ABB RAPID module: ReplayTargets_v13.mod

MODULE ReplayTargets_v13
    ! Generated from tests_v13.csv and success_v13.csv.
    ! Target names include version and testId. B* variants include version, testId, and confId.

    ! Robtargets and jointtargets for replay
    CONST robtarget rA_v13_t1 := [[1867.5,0,1823],[2.18557E-8,0,-1,0],[0,0,0,0],[9E+09,9E+09,9E+09,9E+09,9E+09,9E+09]];
    CONST robtarget rB_v13_t1 := [[99.2091,-1417.11,3170.05],[0.75375,-0.215208,0.229423,-0.576985],[-2,-3,2,0],[9E+09,9E+09,9E+09,9E+09,9E+09,9E+09]];
    CONST robtarget rB_v13_t1_c2 := [[99.2091,-1417.11,3170.05],[0.75375,-0.215208,0.229423,-0.576985],[0,0,-4,0],[9E+09,9E+09,9E+09,9E+09,9E+09,9E+09]];
    CONST jointtarget jA_v13_t1 := [[0,-2.3802E-6,7.25062E-7,0,90,0],[9E+09,9E+09,9E+09,9E+09,9E+09,9E+09]];
    CONST jointtarget jB_v13_t1 := [[-90.0009,9.75799,-56.39,-225.001,57.1728,224.999],[9E+09,9E+09,9E+09,9E+09,9E+09,9E+09]];
    CONST jointtarget jBseed_v13_t1 := [[-90.0009,9.75799,-56.39,-225.001,57.1728,224.999],[9E+09,9E+09,9E+09,9E+09,9E+09,9E+09]];

    CONST robtarget rA_v13_t2 := [[99.2091,-1417.11,3170.05],[0.75375,-0.215208,0.229423,-0.576985],[-2,-3,2,0],[9E+09,9E+09,9E+09,9E+09,9E+09,9E+09]];
    CONST robtarget rB_v13_t2 := [[-1176.87,-1004.25,553.318],[0.0696016,-0.873055,0.122095,0.466929],[-2,3,1,0],[9E+09,9E+09,9E+09,9E+09,9E+09,9E+09]];
    CONST robtarget rB_v13_t2_c5 := [[-1176.87,-1004.25,553.318],[0.0696016,-0.873055,0.122095,0.466929],[0,0,0,0],[9E+09,9E+09,9E+09,9E+09,9E+09,9E+09]];
    CONST jointtarget jA_v13_t2 := [[-90.0009,9.75799,-56.39,-225.001,57.1728,224.999],[9E+09,9E+09,9E+09,9E+09,9E+09,9E+09]];
    CONST jointtarget jB_v13_t2 := [[-134.999,4.65286,49.6707,270.001,46.9753,135.001],[9E+09,9E+09,9E+09,9E+09,9E+09,9E+09]];
    CONST jointtarget jBseed_v13_t2 := [[-134.999,4.65285,49.6707,270.001,46.9753,135.001],[9E+09,9E+09,9E+09,9E+09,9E+09,9E+09]];

    CONST robtarget rA_v13_t3 := [[-1176.87,-1004.25,553.318],[0.0696016,-0.873055,0.122095,0.466929],[-2,3,1,0],[9E+09,9E+09,9E+09,9E+09,9E+09,9E+09]];
    CONST robtarget rB_v13_t3 := [[-0.00217641,-566.482,3480.85],[0.983173,-0.182676,1.08969E-6,-6.64925E-6],[-2,-3,-2,0],[9E+09,9E+09,9E+09,9E+09,9E+09,9E+09]];
    CONST robtarget rB_v13_t3_c8 := [[-0.00217641,-566.482,3480.85],[0.983173,-0.182676,1.08969E-6,-6.64925E-6],[0,0,4,0],[9E+09,9E+09,9E+09,9E+09,9E+09,9E+09]];
    CONST jointtarget jA_v13_t3 := [[-134.999,4.65286,49.6707,270.001,46.9753,135.001],[9E+09,9E+09,9E+09,9E+09,9E+09,9E+09]];
    CONST jointtarget jB_v13_t3 := [[-90.0003,1.44106,-73.8029,-180,38.6896,-90.0003],[9E+09,9E+09,9E+09,9E+09,9E+09,9E+09]];
    CONST jointtarget jBseed_v13_t3 := [[-90.0003,1.44108,-73.8029,-180,38.6895,-90.0003],[9E+09,9E+09,9E+09,9E+09,9E+09,9E+09]];

    CONST robtarget rA_v13_t4 := [[-0.00217641,-566.482,3480.85],[0.983173,-0.182676,1.08969E-6,-6.64925E-6],[-2,-3,-2,0],[9E+09,9E+09,9E+09,9E+09,9E+09,9E+09]];
    CONST robtarget rB_v13_t4 := [[1002.23,-1002.24,1474.39],[0.334755,0.447696,-0.18544,0.808158],[-1,1,-5,0],[9E+09,9E+09,9E+09,9E+09,9E+09,9E+09]];
    CONST robtarget rB_v13_t4_c1 := [[1002.23,-1002.24,1474.39],[0.334755,0.447696,-0.18544,0.808158],[0,-4,-4,0],[9E+09,9E+09,9E+09,9E+09,9E+09,9E+09]];
    CONST robtarget rB_v13_t4_c4 := [[1002.23,-1002.24,1474.39],[0.334755,0.447696,-0.18544,0.808158],[0,-4,0,0],[9E+09,9E+09,9E+09,9E+09,9E+09,9E+09]];
    CONST jointtarget jA_v13_t4 := [[-90.0003,1.44106,-73.8029,-180,38.6896,-90.0003],[9E+09,9E+09,9E+09,9E+09,9E+09,9E+09]];
    CONST jointtarget jB_v13_t4 := [[-45.0002,-31.5629,47.7187,180,48.1857,-360],[9E+09,9E+09,9E+09,9E+09,9E+09,9E+09]];
    CONST jointtarget jBseed_v13_t4 := [[-45.0002,-31.5629,47.7187,180,48.1857,-360],[9E+09,9E+09,9E+09,9E+09,9E+09,9E+09]];

    CONST robtarget rA_v13_t7 := [[-1.66635,-2612.43,1764.4],[0.48959,0.510166,0.505346,-0.494629],[-2,-2,-3,0],[9E+09,9E+09,9E+09,9E+09,9E+09,9E+09]];
    CONST robtarget rB_v13_t7 := [[1079.75,897.425,1506.87],[0.173905,-0.697828,0.271448,-0.639616],[0,-2,-1,0],[9E+09,9E+09,9E+09,9E+09,9E+09,9E+09]];
    CONST robtarget rB_v13_t7_c5 := [[1079.75,897.425,1506.87],[0.173905,-0.697828,0.271448,-0.639616],[0,0,0,0],[9E+09,9E+09,9E+09,9E+09,9E+09,9E+09]];
    CONST jointtarget jA_v13_t7 := [[-90.0005,30.6583,-28.3007,-135.001,0.798362,-225],[9E+09,9E+09,9E+09,9E+09,9E+09,9E+09]];
    CONST jointtarget jB_v13_t7 := [[44.9993,-31.3907,42.3905,-90.0007,50.524,-45.0007],[9E+09,9E+09,9E+09,9E+09,9E+09,9E+09]];
    CONST jointtarget jBseed_v13_t7 := [[44.9993,-31.3907,42.3905,-90.0007,50.524,-45.0007],[9E+09,9E+09,9E+09,9E+09,9E+09,9E+09]];

    CONST robtarget rA_v13_t9 := [[-1827.27,-1738.5,375.985],[0.181266,-0.630243,-0.526884,0.540675],[-2,2,-4,0],[9E+09,9E+09,9E+09,9E+09,9E+09,9E+09]];
    CONST robtarget rB_v13_t9 := [[1928.3,-1922.53,935.585],[0.214413,-0.329221,0.77773,-0.49069],[-1,-3,2,0],[9E+09,9E+09,9E+09,9E+09,9E+09,9E+09]];
    CONST robtarget rB_v13_t9_c2 := [[1928.3,-1922.53,935.585],[0.214413,-0.329221,0.77773,-0.49069],[0,0,-4,0],[9E+09,9E+09,9E+09,9E+09,9E+09,9E+09]];
    CONST jointtarget jA_v13_t9 := [[-135.001,48.6288,-2.55226,224.999,32.0902,-270.001],[9E+09,9E+09,9E+09,9E+09,9E+09,9E+09]];
    CONST jointtarget jB_v13_t9 := [[-44.9999,43.2234,-17.9696,-270,1.39897,180],[9E+09,9E+09,9E+09,9E+09,9E+09,9E+09]];
    CONST jointtarget jBseed_v13_t9 := [[-44.9999,43.2234,-17.9696,-270,1.39897,180],[9E+09,9E+09,9E+09,9E+09,9E+09,9E+09]];

    CONST robtarget rA_v13_t12 := [[-222.385,-252.882,3208.41],[0.390141,0.148006,0.129266,-0.899541],[-2,1,2,0],[9E+09,9E+09,9E+09,9E+09,9E+09,9E+09]];
    CONST robtarget rB_v13_t12 := [[1041.72,97.8898,1906.32],[0.539625,-0.399974,-0.105401,-0.733292],[-1,-3,-4,0],[9E+09,9E+09,9E+09,9E+09,9E+09,9E+09]];
    CONST robtarget rB_v13_t12_c5 := [[1041.72,97.8898,1906.32],[0.539625,-0.399974,-0.105401,-0.733292],[0,0,0,0],[9E+09,9E+09,9E+09,9E+09,9E+09,9E+09]];
    CONST jointtarget jA_v13_t12 := [[-135,-33.5441,-27.4954,135,10.5234,225],[9E+09,9E+09,9E+09,9E+09,9E+09,9E+09]];
    CONST jointtarget jB_v13_t12 := [[-0.000837912,-50.3464,42.4104,-225.001,56.0045,-270.001],[9E+09,9E+09,9E+09,9E+09,9E+09,9E+09]];
    CONST jointtarget jBseed_v13_t12 := [[-0.000838008,-50.3464,42.4104,-225.001,56.0045,-270.001],[9E+09,9E+09,9E+09,9E+09,9E+09,9E+09]];

    CONST robtarget rA_v13_t14 := [[-711.848,-569.761,2198.67],[0.583194,0.0205634,-0.810946,0.0427693],[-2,-1,2,0],[9E+09,9E+09,9E+09,9E+09,9E+09,9E+09]];
    CONST robtarget rB_v13_t14 := [[572.003,-670.137,3433.99],[0.0410544,-0.0140871,-0.281004,0.958725],[-1,3,-1,0],[9E+09,9E+09,9E+09,9E+09,9E+09,9E+09]];
    CONST robtarget rB_v13_t14_c5 := [[572.003,-670.137,3433.99],[0.0410544,-0.0140871,-0.281004,0.958725],[0,0,0,0],[9E+09,9E+09,9E+09,9E+09,9E+09,9E+09]];
    CONST robtarget rB_v13_t14_c8 := [[572.003,-670.137,3433.99],[0.0410544,-0.0140871,-0.281004,0.958725],[0,0,4,0],[9E+09,9E+09,9E+09,9E+09,9E+09,9E+09]];
    CONST jointtarget jA_v13_t14 := [[-135,-49.0756,23.5295,-45.0005,58.2934,225],[9E+09,9E+09,9E+09,9E+09,9E+09,9E+09]];
    CONST jointtarget jB_v13_t14 := [[-44.9991,5.08498,-72.811,270.001,24.557,-44.9991],[9E+09,9E+09,9E+09,9E+09,9E+09,9E+09]];
    CONST jointtarget jBseed_v13_t14 := [[-44.9991,5.085,-72.8111,270.001,24.557,-44.9991],[9E+09,9E+09,9E+09,9E+09,9E+09,9E+09]];

    CONST robtarget rA_v13_t16 := [[1137.15,-8.72496,2432.97],[0.836307,0.0218099,0.54764,-0.0143057],[-1,2,-4,0],[9E+09,9E+09,9E+09,9E+09,9E+09,9E+09]];
    CONST robtarget rB_v13_t16 := [[1938.99,24.0931,2499.76],[0.282343,0.471451,0.258319,0.794536],[0,1,0,0],[9E+09,9E+09,9E+09,9E+09,9E+09,9E+09]];
    CONST robtarget rB_v13_t16_c2 := [[1938.99,24.0931,2499.76],[0.282343,0.471451,0.258319,0.794536],[0,0,-4,0],[9E+09,9E+09,9E+09,9E+09,9E+09,9E+09]];
    CONST robtarget rB_v13_t16_c5 := [[1938.99,24.0931,2499.76],[0.282343,0.471451,0.258319,0.794536],[0,0,0,0],[9E+09,9E+09,9E+09,9E+09,9E+09,9E+09]];
    CONST jointtarget jA_v13_t16 := [[-0.000942424,-37.0122,13.4483,269.999,2.98837,-270.001],[9E+09,9E+09,9E+09,9E+09,9E+09,9E+09]];
    CONST jointtarget jB_v13_t16 := [[2.68408E-5,2.38228,-19.2432,135,11.7722,3.5699E-5],[9E+09,9E+09,9E+09,9E+09,9E+09,9E+09]];
    CONST jointtarget jBseed_v13_t16 := [[2.67647E-5,2.38227,-19.2431,135,11.7722,2.67647E-5],[9E+09,9E+09,9E+09,9E+09,9E+09,9E+09]];

    CONST robtarget rA_v13_t17 := [[1938.99,24.0931,2499.76],[0.282343,0.471451,0.258319,0.794536],[0,1,0,0],[9E+09,9E+09,9E+09,9E+09,9E+09,9E+09]];
    CONST robtarget rB_v13_t17 := [[-0.0282522,-2261.74,5.33349],[0.35869,0.933457,6.24728E-6,-5.58097E-6],[-2,-3,2,0],[9E+09,9E+09,9E+09,9E+09,9E+09,9E+09]];
    CONST robtarget rB_v13_t17_c5 := [[-0.0282522,-2261.74,5.33349],[0.35869,0.933457,6.24728E-6,-5.58097E-6],[0,0,0,0],[9E+09,9E+09,9E+09,9E+09,9E+09,9E+09]];
    CONST jointtarget jA_v13_t17 := [[2.68408E-5,2.38228,-19.2432,135,11.7722,3.5699E-5],[9E+09,9E+09,9E+09,9E+09,9E+09,9E+09]];
    CONST jointtarget jB_v13_t17 := [[-90.0007,51.6062,8.15576,-180.001,11.8015,269.999],[9E+09,9E+09,9E+09,9E+09,9E+09,9E+09]];
    CONST jointtarget jBseed_v13_t17 := [[-90.0007,51.6062,8.15576,-180.001,11.8015,269.999],[9E+09,9E+09,9E+09,9E+09,9E+09,9E+09]];

    CONST robtarget rA_v13_t18 := [[-0.0282522,-2261.74,5.33349],[0.35869,0.933457,6.24728E-6,-5.58097E-6],[-2,-3,2,0],[9E+09,9E+09,9E+09,9E+09,9E+09,9E+09]];
    CONST robtarget rB_v13_t18 := [[-56.7244,-1514.12,2175.5],[0.65245,0.637838,0.121596,-0.390751],[-1,-1,-3,0],[9E+09,9E+09,9E+09,9E+09,9E+09,9E+09]];
    CONST robtarget rB_v13_t18_c5 := [[-56.7244,-1514.12,2175.5],[0.65245,0.637838,0.121596,-0.390751],[0,0,0,0],[9E+09,9E+09,9E+09,9E+09,9E+09,9E+09]];
    CONST jointtarget jA_v13_t18 := [[-90.0007,51.6062,8.15576,-180.001,11.8015,269.999],[9E+09,9E+09,9E+09,9E+09,9E+09,9E+09]];
    CONST jointtarget jB_v13_t18 := [[-89.9991,-23.8722,14.2775,-89.9991,19.8657,-224.999],[9E+09,9E+09,9E+09,9E+09,9E+09,9E+09]];
    CONST jointtarget jBseed_v13_t18 := [[-89.9991,-23.8722,14.2775,-89.9991,19.8657,-224.999],[9E+09,9E+09,9E+09,9E+09,9E+09,9E+09]];

    CONST robtarget rA_v13_t21 := [[1261.7,1309.55,913.586],[0.285378,-0.764589,-0.364994,-0.448043],[0,-3,-4,0],[9E+09,9E+09,9E+09,9E+09,9E+09,9E+09]];
    CONST robtarget rB_v13_t21 := [[93.0833,-128.762,3074.48],[0.882421,0.41568,0.199326,-0.0938791],[0,3,1,0],[9E+09,9E+09,9E+09,9E+09,9E+09,9E+09]];
    CONST robtarget rB_v13_t21_c2 := [[93.0833,-128.762,3074.48],[0.882421,0.41568,0.199326,-0.0938791],[0,0,-4,0],[9E+09,9E+09,9E+09,9E+09,9E+09,9E+09]];
    CONST jointtarget jA_v13_t21 := [[44.9995,0.72329,37.6376,-225,16.6576,-315],[9E+09,9E+09,9E+09,9E+09,9E+09,9E+09]];
    CONST jointtarget jB_v13_t21 := [[0.000667693,-42.5385,-22.0045,270.001,50.4471,90.0007],[9E+09,9E+09,9E+09,9E+09,9E+09,9E+09]];
    CONST jointtarget jBseed_v13_t21 := [[0.000663381,-42.5385,-22.0045,270.001,50.4471,90.0007],[9E+09,9E+09,9E+09,9E+09,9E+09,9E+09]];

    CONST robtarget rA_v13_t22 := [[93.0833,-128.762,3074.48],[0.882421,0.41568,0.199326,-0.0938791],[0,3,1,0],[9E+09,9E+09,9E+09,9E+09,9E+09,9E+09]];
    CONST robtarget rB_v13_t22 := [[289.912,345.963,3026.72],[0.857655,-0.223007,0.2415,0.39544],[0,0,2,0],[9E+09,9E+09,9E+09,9E+09,9E+09,9E+09]];
    CONST robtarget rB_v13_t22_c8 := [[289.912,345.963,3026.72],[0.857655,-0.223007,0.2415,0.39544],[0,0,4,0],[9E+09,9E+09,9E+09,9E+09,9E+09,9E+09]];
    CONST jointtarget jA_v13_t22 := [[0.000667693,-42.5385,-22.0045,270.001,50.4471,90.0007],[9E+09,9E+09,9E+09,9E+09,9E+09,9E+09]];
    CONST jointtarget jB_v13_t22 := [[44.9997,-39.9237,-13.8752,89.9997,13.7297,270],[9E+09,9E+09,9E+09,9E+09,9E+09,9E+09]];
    CONST jointtarget jBseed_v13_t22 := [[44.9997,-39.9237,-13.8752,89.9997,13.7297,270],[9E+09,9E+09,9E+09,9E+09,9E+09,9E+09]];

    CONST robtarget rA_v13_t23 := [[289.912,345.963,3026.72],[0.857655,-0.223007,0.2415,0.39544],[0,0,2,0],[9E+09,9E+09,9E+09,9E+09,9E+09,9E+09]];
    CONST robtarget rB_v13_t23 := [[1448.72,1285.3,532.252],[0.149019,-0.761761,0.449066,-0.442553],[0,-2,-5,0],[9E+09,9E+09,9E+09,9E+09,9E+09,9E+09]];
    CONST robtarget rB_v13_t23_c9 := [[1448.72,1285.3,532.252],[0.149019,-0.761761,0.449066,-0.442553],[0,4,4,0],[9E+09,9E+09,9E+09,9E+09,9E+09,9E+09]];
    CONST jointtarget jA_v13_t23 := [[44.9997,-39.9237,-13.8752,89.9997,13.7297,270],[9E+09,9E+09,9E+09,9E+09,9E+09,9E+09]];
    CONST jointtarget jB_v13_t23 := [[45,21.7664,29.5877,-90,43.7819,-360],[9E+09,9E+09,9E+09,9E+09,9E+09,9E+09]];
    CONST jointtarget jBseed_v13_t23 := [[45,21.7664,29.5877,-90,43.7819,-360],[9E+09,9E+09,9E+09,9E+09,9E+09,9E+09]];

    CONST robtarget rA_v13_t25 := [[1386.04,-107.763,3007.42],[0.497407,-0.0630243,0.502569,-0.7043],[-1,2,-1,0],[9E+09,9E+09,9E+09,9E+09,9E+09,9E+09]];
    CONST robtarget rB_v13_t25 := [[1396.9,1402.69,1993.46],[0.265925,0.259196,0.648363,0.664625],[0,1,-1,0],[9E+09,9E+09,9E+09,9E+09,9E+09,9E+09]];
    CONST robtarget rB_v13_t25_c5 := [[1396.9,1402.69,1993.46],[0.265925,0.259196,0.648363,0.664625],[0,0,0,0],[9E+09,9E+09,9E+09,9E+09,9E+09,9E+09]];
    CONST jointtarget jA_v13_t25 := [[-0.000473063,-4.98611,-34.6049,270,40.1819,-0.000475164],[9E+09,9E+09,9E+09,9E+09,9E+09,9E+09]];
    CONST jointtarget jB_v13_t25 := [[45.0004,-2.79976,2.77596,135,1.98309,-44.9996],[9E+09,9E+09,9E+09,9E+09,9E+09,9E+09]];
    CONST jointtarget jBseed_v13_t25 := [[45.0004,-2.79977,2.77596,135,1.98309,-44.9996],[9E+09,9E+09,9E+09,9E+09,9E+09,9E+09]];

    CONST robtarget rA_v13_t26 := [[1396.9,1402.69,1993.46],[0.265925,0.259196,0.648363,0.664625],[0,1,-1,0],[9E+09,9E+09,9E+09,9E+09,9E+09,9E+09]];
    CONST robtarget rB_v13_t26 := [[992.793,-1120.03,211.35],[0.312884,0.309441,-0.897953,0.00551771],[-1,-1,-1,0],[9E+09,9E+09,9E+09,9E+09,9E+09,9E+09]];
    CONST robtarget rB_v13_t26_c5 := [[992.793,-1120.03,211.35],[0.312884,0.309441,-0.897953,0.00551771],[0,0,0,0],[9E+09,9E+09,9E+09,9E+09,9E+09,9E+09]];
    CONST jointtarget jA_v13_t26 := [[45.0004,-2.79976,2.77596,135,1.98309,-44.9996],[9E+09,9E+09,9E+09,9E+09,9E+09,9E+09]];
    CONST jointtarget jB_v13_t26 := [[-44.9994,23.1617,44.406,-44.9994,49.6451,-44.9994],[9E+09,9E+09,9E+09,9E+09,9E+09,9E+09]];
    CONST jointtarget jBseed_v13_t26 := [[-44.9994,23.1617,44.406,-44.9994,49.6451,-44.9994],[9E+09,9E+09,9E+09,9E+09,9E+09,9E+09]];

    CONST robtarget rA_v13_t27 := [[992.793,-1120.03,211.35],[0.312884,0.309441,-0.897953,0.00551771],[-1,-1,-1,0],[9E+09,9E+09,9E+09,9E+09,9E+09,9E+09]];
    CONST robtarget rB_v13_t27 := [[-0.00100132,-1466.24,3231.41],[0.915589,-0.123492,-0.0511516,-0.37925],[-2,1,2,0],[9E+09,9E+09,9E+09,9E+09,9E+09,9E+09]];
    CONST robtarget rB_v13_t27_c1 := [[-0.00100132,-1466.24,3231.41],[0.915589,-0.123492,-0.0511516,-0.37925],[0,-4,-4,0],[9E+09,9E+09,9E+09,9E+09,9E+09,9E+09]];
    CONST robtarget rB_v13_t27_c2 := [[-0.00100132,-1466.24,3231.41],[0.915589,-0.123492,-0.0511516,-0.37925],[0,0,-4,0],[9E+09,9E+09,9E+09,9E+09,9E+09,9E+09]];
    CONST jointtarget jA_v13_t27 := [[-44.9994,23.1617,44.406,-44.9994,49.6451,-44.9994],[9E+09,9E+09,9E+09,9E+09,9E+09,9E+09]];
    CONST jointtarget jB_v13_t27 := [[-90,24.5424,-79.4803,180,50.4251,225],[9E+09,9E+09,9E+09,9E+09,9E+09,9E+09]];
    CONST jointtarget jBseed_v13_t27 := [[-90,24.5424,-79.4803,180,50.4251,225],[9E+09,9E+09,9E+09,9E+09,9E+09,9E+09]];

    CONST robtarget rA_v13_t28 := [[-0.00100132,-1466.24,3231.41],[0.915589,-0.123492,-0.0511516,-0.37925],[-2,1,2,0],[9E+09,9E+09,9E+09,9E+09,9E+09,9E+09]];
    CONST robtarget rB_v13_t28 := [[1759.52,-84.0859,432.636],[0.169271,-0.529813,0.629971,-0.542017],[0,2,-4,0],[9E+09,9E+09,9E+09,9E+09,9E+09,9E+09]];
    CONST robtarget rB_v13_t28_c6 := [[1759.52,-84.0859,432.636],[0.169271,-0.529813,0.629971,-0.542017],[0,4,0,0],[9E+09,9E+09,9E+09,9E+09,9E+09,9E+09]];
    CONST jointtarget jA_v13_t28 := [[-90,24.5424,-79.4803,180,50.4251,225],[9E+09,9E+09,9E+09,9E+09,9E+09,9E+09]];
    CONST jointtarget jB_v13_t28 := [[0.000217785,18.7121,41.2082,225,45.4079,-315],[9E+09,9E+09,9E+09,9E+09,9E+09,9E+09]];
    CONST jointtarget jBseed_v13_t28 := [[0.000217933,18.7121,41.2082,225,45.4079,-315],[9E+09,9E+09,9E+09,9E+09,9E+09,9E+09]];

    CONST robtarget rA_v13_t30 := [[1284.9,1168.38,866.12],[0.010138,-0.726367,-0.185371,-0.66176],[0,-2,3,0],[9E+09,9E+09,9E+09,9E+09,9E+09,9E+09]];
    CONST robtarget rB_v13_t30 := [[-1445.04,1445.04,658.393],[0.0286784,0.921282,-0.381607,0.0692355],[1,0,-4,0],[9E+09,9E+09,9E+09,9E+09,9E+09,9E+09]];
    CONST robtarget rB_v13_t30_c8 := [[-1445.04,1445.04,658.393],[0.0286784,0.921282,-0.381607,0.0692355],[0,0,4,0],[9E+09,9E+09,9E+09,9E+09,9E+09,9E+09]];
    CONST jointtarget jA_v13_t30 := [[44.9991,-0.0750814,42.8071,-135.001,44.2286,314.999],[9E+09,9E+09,9E+09,9E+09,9E+09,9E+09]];
    CONST jointtarget jB_v13_t30 := [[135,23.8905,17.384,1.67051E-5,57.3211,-360],[9E+09,9E+09,9E+09,9E+09,9E+09,9E+09]];
    CONST jointtarget jBseed_v13_t30 := [[135,23.8905,17.384,1.68767E-5,57.3211,-360],[9E+09,9E+09,9E+09,9E+09,9E+09,9E+09]];

    CONST robtarget rA_v13_t34 := [[748.242,-941.627,2112.58],[0.692779,0.646669,0.137038,-0.288266],[-1,2,-3,0],[9E+09,9E+09,9E+09,9E+09,9E+09,9E+09]];
    CONST robtarget rB_v13_t34 := [[2649.92,104.837,1638.1],[0.470426,-0.728833,0.0588047,-0.494008],[0,1,-3,0],[9E+09,9E+09,9E+09,9E+09,9E+09,9E+09]];
    CONST robtarget rB_v13_t34_c2 := [[2649.92,104.837,1638.1],[0.470426,-0.728833,0.0588047,-0.494008],[0,0,-4,0],[9E+09,9E+09,9E+09,9E+09,9E+09,9E+09]];
    CONST jointtarget jA_v13_t34 := [[-45.0002,-37.6678,24.9815,270,54.9644,-225],[9E+09,9E+09,9E+09,9E+09,9E+09,9E+09]];
    CONST jointtarget jB_v13_t34 := [[0.000542358,34.9284,-29.8202,90.0005,38.8745,-224.999],[9E+09,9E+09,9E+09,9E+09,9E+09,9E+09]];
    CONST jointtarget jBseed_v13_t34 := [[0.000542222,34.9284,-29.8202,90.0005,38.8745,-224.999],[9E+09,9E+09,9E+09,9E+09,9E+09,9E+09]];

    CONST robtarget rA_v13_t40 := [[88.1653,-2304.04,1942.16],[0.3419,0.618964,-0.345048,0.617195],[-2,-4,0,0],[9E+09,9E+09,9E+09,9E+09,9E+09,9E+09]];
    CONST robtarget rB_v13_t40 := [[52.8599,-2411.7,1286.37],[0.133416,0.358674,-0.630122,0.675647],[-2,-3,-4,0],[9E+09,9E+09,9E+09,9E+09,9E+09,9E+09]];
    CONST robtarget rB_v13_t40_c4 := [[52.8599,-2411.7,1286.37],[0.133416,0.358674,-0.630122,0.675647],[0,-4,0,0],[9E+09,9E+09,9E+09,9E+09,9E+09,9E+09]];
    CONST jointtarget jA_v13_t40 := [[-90.0007,15.2037,-14.9107,-270.001,31.8778,89.9993],[9E+09,9E+09,9E+09,9E+09,9E+09,9E+09]];
    CONST jointtarget jB_v13_t40 := [[-90.0001,22.4659,0.133673,-225,26.5932,-270],[9E+09,9E+09,9E+09,9E+09,9E+09,9E+09]];
    CONST jointtarget jBseed_v13_t40 := [[-90.0001,22.4659,0.133675,-225,26.5932,-270],[9E+09,9E+09,9E+09,9E+09,9E+09,9E+09]];

    CONST robtarget rA_v13_t41 := [[52.8599,-2411.7,1286.37],[0.133416,0.358674,-0.630122,0.675647],[-2,-3,-4,0],[9E+09,9E+09,9E+09,9E+09,9E+09,9E+09]];
    CONST robtarget rB_v13_t41 := [[2632.93,-42.8013,917.401],[0.298222,0.810035,0.263286,0.430798],[-1,3,2,0],[9E+09,9E+09,9E+09,9E+09,9E+09,9E+09]];
    CONST robtarget rB_v13_t41_c2 := [[2632.93,-42.8013,917.401],[0.298222,0.810035,0.263286,0.430798],[0,0,-4,0],[9E+09,9E+09,9E+09,9E+09,9E+09,9E+09]];
    CONST jointtarget jA_v13_t41 := [[-90.0001,22.4659,0.133673,-225,26.5932,-270],[9E+09,9E+09,9E+09,9E+09,9E+09,9E+09]];
    CONST jointtarget jB_v13_t41 := [[-1.40126E-6,39.2132,-11.4036,270,14.8503,225],[9E+09,9E+09,9E+09,9E+09,9E+09,9E+09]];
    CONST jointtarget jBseed_v13_t41 := [[-1.43435E-6,39.2132,-11.4035,270,14.8503,225],[9E+09,9E+09,9E+09,9E+09,9E+09,9E+09]];

    CONST robtarget rA_v13_t43 := [[-82.306,-1263.49,2466.69],[0.533736,0.754108,0.0698941,-0.376246],[-1,-1,1,0],[9E+09,9E+09,9E+09,9E+09,9E+09,9E+09]];
    CONST robtarget rB_v13_t43 := [[1500.95,-0.00864055,2131.2],[0.68854,-1.66573E-6,0.725198,-6.29854E-6],[-1,-1,-5,0],[9E+09,9E+09,9E+09,9E+09,9E+09,9E+09]];
    CONST robtarget rB_v13_t43_c5 := [[1500.95,-0.00864055,2131.2],[0.68854,-1.66573E-6,0.725198,-6.29854E-6],[0,0,0,0],[9E+09,9E+09,9E+09,9E+09,9E+09,9E+09]];
    CONST jointtarget jA_v13_t43 := [[-90,-27.7285,2.96243,-45,44.1865,90],[9E+09,9E+09,9E+09,9E+09,9E+09,9E+09]];
    CONST jointtarget jB_v13_t43 := [[-0.000322001,-25.2528,15.5907,-0.000322001,12.6328,-360],[9E+09,9E+09,9E+09,9E+09,9E+09,9E+09]];
    CONST jointtarget jBseed_v13_t43 := [[-0.000322001,-25.2528,15.5907,-0.000322001,12.6328,-360],[9E+09,9E+09,9E+09,9E+09,9E+09,9E+09]];

    CONST robtarget rA_v13_t46 := [[-1039.26,-950.35,3214.73],[0.0696838,-0.241685,0.0171566,0.967697],[-2,2,0,0],[9E+09,9E+09,9E+09,9E+09,9E+09,9E+09]];
    CONST robtarget rB_v13_t46 := [[2557.04,-0.0208453,729.575],[0.463781,-0.533766,0.53376,-0.46379],[-1,-3,-4,0],[9E+09,9E+09,9E+09,9E+09,9E+09,9E+09]];
    CONST robtarget rB_v13_t46_c5 := [[2557.04,-0.0208453,729.575],[0.463781,-0.533766,0.53376,-0.46379],[0,0,0,0],[9E+09,9E+09,9E+09,9E+09,9E+09,9E+09]];
    CONST jointtarget jA_v13_t46 := [[-135.001,8.22718,-56.5526,224.999,32.158,89.9992],[9E+09,9E+09,9E+09,9E+09,9E+09,9E+09]];
    CONST jointtarget jB_v13_t46 := [[-0.000482548,39.8871,-2.67922,-180,29.1824,-270],[9E+09,9E+09,9E+09,9E+09,9E+09,9E+09]];
    CONST jointtarget jBseed_v13_t46 := [[-0.000482467,39.8871,-2.67921,-180,29.1824,-270],[9E+09,9E+09,9E+09,9E+09,9E+09,9E+09]];

    CONST robtarget rA_v13_t48 := [[-1863.63,1884.03,577.956],[0.137672,0.322591,-0.830191,-0.433319],[1,-1,-2,0],[9E+09,9E+09,9E+09,9E+09,9E+09,9E+09]];
    CONST robtarget rB_v13_t48 := [[-1714.66,1743.11,2527.4],[0.805088,-0.490131,-0.146718,0.300131],[1,3,0,0],[9E+09,9E+09,9E+09,9E+09,9E+09,9E+09]];
    CONST robtarget rB_v13_t48_c2 := [[-1714.66,1743.11,2527.4],[0.805088,-0.490131,-0.146718,0.300131],[0,0,-4,0],[9E+09,9E+09,9E+09,9E+09,9E+09,9E+09]];
    CONST robtarget rB_v13_t48_c3 := [[-1714.66,1743.11,2527.4],[0.805088,-0.490131,-0.146718,0.300131],[0,4,-4,0],[9E+09,9E+09,9E+09,9E+09,9E+09,9E+09]];
    CONST jointtarget jA_v13_t48 := [[135.001,47.5887,-11.5186,-89.9992,4.96963,-179.999],[9E+09,9E+09,9E+09,9E+09,9E+09,9E+09]];
    CONST jointtarget jB_v13_t48 := [[135.001,39.8724,-68.558,270.001,6.93258,0.000757349],[9E+09,9E+09,9E+09,9E+09,9E+09,9E+09]];
    CONST jointtarget jBseed_v13_t48 := [[135.001,39.8724,-68.558,270.001,6.93258,0.000879635],[9E+09,9E+09,9E+09,9E+09,9E+09,9E+09]];

    CONST robtarget rA_v13_t49 := [[-1714.66,1743.11,2527.4],[0.805088,-0.490131,-0.146718,0.300131],[1,3,0,0],[9E+09,9E+09,9E+09,9E+09,9E+09,9E+09]];
    CONST robtarget rB_v13_t49 := [[-92.445,1856.02,295.842],[0.241258,0.732303,-0.611889,-0.176405],[0,0,-1,0],[9E+09,9E+09,9E+09,9E+09,9E+09,9E+09]];
    CONST robtarget rB_v13_t49_c5 := [[-92.445,1856.02,295.842],[0.241258,0.732303,-0.611889,-0.176405],[0,0,0,0],[9E+09,9E+09,9E+09,9E+09,9E+09,9E+09]];
    CONST jointtarget jA_v13_t49 := [[135.001,39.8724,-68.558,270.001,6.93258,0.000757349],[9E+09,9E+09,9E+09,9E+09,9E+09,9E+09]];
    CONST jointtarget jB_v13_t49 := [[89.9998,30.347,27.4889,44.9998,51.5293,-45.0002],[9E+09,9E+09,9E+09,9E+09,9E+09,9E+09]];
    CONST jointtarget jBseed_v13_t49 := [[89.9998,30.347,27.4889,44.9998,51.5293,-45.0002],[9E+09,9E+09,9E+09,9E+09,9E+09,9E+09]];

    CONST robtarget rA_v13_t50 := [[-92.445,1856.02,295.842],[0.241258,0.732303,-0.611889,-0.176405],[0,0,-1,0],[9E+09,9E+09,9E+09,9E+09,9E+09,9E+09]];
    CONST robtarget rB_v13_t50 := [[59.5501,2247.64,2712.96],[0.410824,-0.0300862,0.490117,0.768182],[0,2,-3,0],[9E+09,9E+09,9E+09,9E+09,9E+09,9E+09]];
    CONST robtarget rB_v13_t50_c3 := [[59.5501,2247.64,2712.96],[0.410824,-0.0300862,0.490117,0.768182],[0,4,-4,0],[9E+09,9E+09,9E+09,9E+09,9E+09,9E+09]];
    CONST jointtarget jA_v13_t50 := [[89.9998,30.347,27.4889,44.9998,51.5293,-45.0002],[9E+09,9E+09,9E+09,9E+09,9E+09,9E+09]];
    CONST jointtarget jB_v13_t50 := [[89.9995,33.6393,-67.2924,270,20.8838,-225.001],[9E+09,9E+09,9E+09,9E+09,9E+09,9E+09]];
    CONST jointtarget jBseed_v13_t50 := [[89.9995,33.6393,-67.2924,270,20.8838,-225],[9E+09,9E+09,9E+09,9E+09,9E+09,9E+09]];

    CONST robtarget rA_v13_t52 := [[744.455,559.841,3380.27],[0.685218,0.425237,0.178412,0.563754],[0,-1,1,0],[9E+09,9E+09,9E+09,9E+09,9E+09,9E+09]];
    CONST robtarget rB_v13_t52 := [[897.628,-24.8198,3391.83],[0.0188222,0.17807,-0.072298,0.981178],[-1,2,-1,0],[9E+09,9E+09,9E+09,9E+09,9E+09,9E+09]];
    CONST robtarget rB_v13_t52_c7 := [[897.628,-24.8198,3391.83],[0.0188222,0.17807,-0.072298,0.981178],[0,-4,4,0],[9E+09,9E+09,9E+09,9E+09,9E+09,9E+09]];
    CONST jointtarget jA_v13_t52 := [[45.0007,7.46181,-74.6202,-89.9993,51.4212,135.001],[9E+09,9E+09,9E+09,9E+09,9E+09,9E+09]];
    CONST jointtarget jB_v13_t52 := [[-0.000498019,-3.05978,-57.7746,225,12.1293,-45.0005],[9E+09,9E+09,9E+09,9E+09,9E+09,9E+09]];
    CONST jointtarget jBseed_v13_t52 := [[-0.000497971,-3.05978,-57.7746,224.999,12.1293,-45.0005],[9E+09,9E+09,9E+09,9E+09,9E+09,9E+09]];

    CONST robtarget rA_v13_t55 := [[35.4897,1052.12,3269.72],[0.908868,-0.402983,0.102442,-0.0326873],[1,-1,-1,0],[9E+09,9E+09,9E+09,9E+09,9E+09,9E+09]];
    CONST robtarget rB_v13_t55 := [[-1776.81,1609.28,356.308],[0.171575,-0.741953,-0.45782,0.458769],[1,-4,1,0],[9E+09,9E+09,9E+09,9E+09,9E+09,9E+09]];
    CONST robtarget rB_v13_t55_c2 := [[-1776.81,1609.28,356.308],[0.171575,-0.741953,-0.45782,0.458769],[0,0,-4,0],[9E+09,9E+09,9E+09,9E+09,9E+09,9E+09]];
    CONST jointtarget jA_v13_t55 := [[90.0005,-6.28621,-48.3084,-44.9995,17.4944,-44.9995],[9E+09,9E+09,9E+09,9E+09,9E+09,9E+09]];
    CONST jointtarget jB_v13_t55 := [[135,45.8236,1.7484,-270,45.1918,180],[9E+09,9E+09,9E+09,9E+09,9E+09,9E+09]];
    CONST jointtarget jBseed_v13_t55 := [[135,45.8235,1.74841,-270,45.1918,180],[9E+09,9E+09,9E+09,9E+09,9E+09,9E+09]];

    CONST robtarget rA_v13_t57 := [[2362.83,-117.08,1981.63],[0.497836,0.697972,-0.00591765,0.514742],[-1,-2,2,0],[9E+09,9E+09,9E+09,9E+09,9E+09,9E+09]];
    CONST robtarget rB_v13_t57 := [[1030.09,969.545,2370.36],[0.765563,-0.413941,0.283798,-0.402522],[0,2,0,0],[9E+09,9E+09,9E+09,9E+09,9E+09,9E+09]];
    CONST robtarget rB_v13_t57_c4 := [[1030.09,969.545,2370.36],[0.765563,-0.413941,0.283798,-0.402522],[0,-4,0,0],[9E+09,9E+09,9E+09,9E+09,9E+09,9E+09]];
    CONST jointtarget jA_v13_t57 := [[-0.000145643,20.0781,-22.1354,-90.0001,44.5106,225],[9E+09,9E+09,9E+09,9E+09,9E+09,9E+09]];
    CONST jointtarget jB_v13_t57 := [[44.9996,-25.5019,9.98871,225,21.25,44.9996],[9E+09,9E+09,9E+09,9E+09,9E+09,9E+09]];
    CONST jointtarget jBseed_v13_t57 := [[44.9996,-25.5019,9.98871,225,21.25,44.9996],[9E+09,9E+09,9E+09,9E+09,9E+09,9E+09]];

    CONST robtarget rA_v13_t58 := [[1030.09,969.545,2370.36],[0.765563,-0.413941,0.283798,-0.402522],[0,2,0,0],[9E+09,9E+09,9E+09,9E+09,9E+09,9E+09]];
    CONST robtarget rB_v13_t58 := [[1171.23,1171.21,2060.9],[0.870528,-0.3094,0.128153,-0.360596],[0,1,-4,0],[9E+09,9E+09,9E+09,9E+09,9E+09,9E+09]];
    CONST robtarget rB_v13_t58_c5 := [[1171.23,1171.21,2060.9],[0.870528,-0.3094,0.128153,-0.360596],[0,0,0,0],[9E+09,9E+09,9E+09,9E+09,9E+09,9E+09]];
    CONST jointtarget jA_v13_t58 := [[44.9996,-25.5019,9.98871,225,21.25,44.9996],[9E+09,9E+09,9E+09,9E+09,9E+09,9E+09]];
    CONST jointtarget jB_v13_t58 := [[44.9994,-16.5001,16.9634,179.999,51.3315,-270.001],[9E+09,9E+09,9E+09,9E+09,9E+09,9E+09]];
    CONST jointtarget jBseed_v13_t58 := [[44.9994,-16.5001,16.9634,179.999,51.3315,-270.001],[9E+09,9E+09,9E+09,9E+09,9E+09,9E+09]];

    CONST robtarget rA_v13_t59 := [[1171.23,1171.21,2060.9],[0.870528,-0.3094,0.128153,-0.360596],[0,1,-4,0],[9E+09,9E+09,9E+09,9E+09,9E+09,9E+09]];
    CONST robtarget rB_v13_t59 := [[607.458,607.447,2147.09],[0.83273,-0.165751,0.40015,0.344916],[0,1,1,0],[9E+09,9E+09,9E+09,9E+09,9E+09,9E+09]];
    CONST robtarget rB_v13_t59_c2 := [[607.458,607.447,2147.09],[0.83273,-0.165751,0.40015,0.344916],[0,0,-4,0],[9E+09,9E+09,9E+09,9E+09,9E+09,9E+09]];
    CONST jointtarget jA_v13_t59 := [[44.9994,-16.5001,16.9634,179.999,51.3315,-270.001],[9E+09,9E+09,9E+09,9E+09,9E+09,9E+09]];
    CONST jointtarget jB_v13_t59 := [[44.9995,-57.6672,35.3047,179.999,16.306,179.999],[9E+09,9E+09,9E+09,9E+09,9E+09,9E+09]];
    CONST jointtarget jBseed_v13_t59 := [[44.9995,-57.6672,35.3047,179.999,16.306,179.999],[9E+09,9E+09,9E+09,9E+09,9E+09,9E+09]];

    CONST robtarget rA_v13_t60 := [[607.458,607.447,2147.09],[0.83273,-0.165751,0.40015,0.344916],[0,1,1,0],[9E+09,9E+09,9E+09,9E+09,9E+09,9E+09]];
    CONST robtarget rB_v13_t60 := [[130.648,1890.82,1987.21],[0.667553,-0.233153,0.66755,0.233218],[1,3,1,0],[9E+09,9E+09,9E+09,9E+09,9E+09,9E+09]];
    CONST robtarget rB_v13_t60_c6 := [[130.648,1890.82,1987.21],[0.667553,-0.233153,0.66755,0.233218],[0,4,0,0],[9E+09,9E+09,9E+09,9E+09,9E+09,9E+09]];
    CONST jointtarget jA_v13_t60 := [[44.9995,-57.6672,35.3047,179.999,16.306,179.999],[9E+09,9E+09,9E+09,9E+09,9E+09,9E+09]];
    CONST jointtarget jB_v13_t60 := [[90.0009,-4.12915,4.12488,270.001,51.4908,90.0009],[9E+09,9E+09,9E+09,9E+09,9E+09,9E+09]];
    CONST jointtarget jBseed_v13_t60 := [[90.0009,-4.12915,4.12488,270.001,51.4908,90.0009],[9E+09,9E+09,9E+09,9E+09,9E+09,9E+09]];

    CONST robtarget rA_v13_t64 := [[1415.95,-1415.95,2149.12],[0.44547,0.809388,0.335259,0.184521],[-1,0,1,0],[9E+09,9E+09,9E+09,9E+09,9E+09,9E+09]];
    CONST robtarget rB_v13_t64 := [[1197.82,-1176.59,2036.72],[0.317237,-0.280893,0.59291,-0.684775],[-1,-3,-3,0],[9E+09,9E+09,9E+09,9E+09,9E+09,9E+09]];
    CONST robtarget rB_v13_t64_c4 := [[1197.82,-1176.59,2036.72],[0.317237,-0.280893,0.59291,-0.684775],[0,-4,0,0],[9E+09,9E+09,9E+09,9E+09,9E+09,9E+09]];
    CONST robtarget rB_v13_t64_c5 := [[1197.82,-1176.59,2036.72],[0.317237,-0.280893,0.59291,-0.684775],[0,0,0,0],[9E+09,9E+09,9E+09,9E+09,9E+09,9E+09]];
    CONST jointtarget jA_v13_t64 := [[-44.9999,2.41157,-11.7884,6.13466E-5,41.7219,90.0001],[9E+09,9E+09,9E+09,9E+09,9E+09,9E+09]];
    CONST jointtarget jB_v13_t64 := [[-44.9997,-17.7453,14.8924,-225,7.30064,-225],[9E+09,9E+09,9E+09,9E+09,9E+09,9E+09]];
    CONST jointtarget jBseed_v13_t64 := [[-44.9997,-17.7453,14.8924,-225,7.30064,-225],[9E+09,9E+09,9E+09,9E+09,9E+09,9E+09]];

    CONST robtarget rA_v13_t68 := [[1236.34,1111.35,2995.76],[0.222181,-0.478252,0.0706308,-0.846713],[0,-2,2,0],[9E+09,9E+09,9E+09,9E+09,9E+09,9E+09]];
    CONST robtarget rB_v13_t68 := [[-57.7184,1820.6,1382.64],[0.148015,0.0998489,-0.702265,-0.689163],[1,-3,-1,0],[9E+09,9E+09,9E+09,9E+09,9E+09,9E+09]];
    CONST robtarget rB_v13_t68_c7 := [[-57.7184,1820.6,1382.64],[0.148015,0.0998489,-0.702265,-0.689163],[0,-4,4,0],[9E+09,9E+09,9E+09,9E+09,9E+09,9E+09]];
    CONST jointtarget jA_v13_t68 := [[44.9997,7.72545,-46.6024,-90.0003,31.9492,270],[9E+09,9E+09,9E+09,9E+09,9E+09,9E+09]];
    CONST jointtarget jB_v13_t68 := [[90.0006,-8.52015,30.5081,-224.999,29.2502,-44.9994],[9E+09,9E+09,9E+09,9E+09,9E+09,9E+09]];
    CONST jointtarget jBseed_v13_t68 := [[90.0006,-8.52016,30.5081,-224.999,29.2502,-44.9994],[9E+09,9E+09,9E+09,9E+09,9E+09,9E+09]];

    CONST robtarget rA_v13_t72 := [[3.5228,3.52427,2875.76],[0.694537,0.187659,-2.73543E-6,-0.694552],[0,-3,0,0],[9E+09,9E+09,9E+09,9E+09,9E+09,9E+09]];
    CONST robtarget rB_v13_t72 := [[63.9337,654.94,3178.75],[0.923073,-0.0384418,0.220425,0.312844],[1,2,-3,0],[9E+09,9E+09,9E+09,9E+09,9E+09,9E+09]];
    CONST robtarget rB_v13_t72_c2 := [[63.9337,654.94,3178.75],[0.923073,-0.0384418,0.220425,0.312844],[0,0,-4,0],[9E+09,9E+09,9E+09,9E+09,9E+09,9E+09]];
    CONST robtarget rB_v13_t72_c5 := [[63.9337,654.94,3178.75],[0.923073,-0.0384418,0.220425,0.312844],[0,0,0,0],[9E+09,9E+09,9E+09,9E+09,9E+09,9E+09]];
    CONST jointtarget jA_v13_t72 := [[44.9995,-55.1842,-2.1833,-180,54.265,44.9995],[9E+09,9E+09,9E+09,9E+09,9E+09,9E+09]];
    CONST jointtarget jB_v13_t72 := [[90.0007,-25.6374,-26.809,225.001,32.7842,-269.999],[9E+09,9E+09,9E+09,9E+09,9E+09,9E+09]];
    CONST jointtarget jBseed_v13_t72 := [[90.0007,-25.6374,-26.809,225.001,32.7842,-269.999],[9E+09,9E+09,9E+09,9E+09,9E+09,9E+09]];

    CONST robtarget rA_v13_t73 := [[63.9337,654.94,3178.75],[0.923073,-0.0384418,0.220425,0.312844],[1,2,-3,0],[9E+09,9E+09,9E+09,9E+09,9E+09,9E+09]];
    CONST robtarget rB_v13_t73 := [[1346.82,1377.44,2243.56],[0.715342,-0.61979,0.203463,-0.2505],[0,-3,2,0],[9E+09,9E+09,9E+09,9E+09,9E+09,9E+09]];
    CONST robtarget rB_v13_t73_c2 := [[1346.82,1377.44,2243.56],[0.715342,-0.61979,0.203463,-0.2505],[0,0,-4,0],[9E+09,9E+09,9E+09,9E+09,9E+09,9E+09]];
    CONST jointtarget jA_v13_t73 := [[90.0007,-25.6374,-26.809,225.001,32.7842,-269.999],[9E+09,9E+09,9E+09,9E+09,9E+09,9E+09]];
    CONST jointtarget jB_v13_t73 := [[45.0008,-2.93161,-5.70633,-269.999,7.44163,180.001],[9E+09,9E+09,9E+09,9E+09,9E+09,9E+09]];
    CONST jointtarget jBseed_v13_t73 := [[45.0008,-2.93161,-5.70634,-269.999,7.44163,180.001],[9E+09,9E+09,9E+09,9E+09,9E+09,9E+09]];

    CONST robtarget rA_v13_t75 := [[54.7805,2533.42,395.018],[0.168511,-0.908383,-0.300909,-0.236427],[1,-1,3,0],[9E+09,9E+09,9E+09,9E+09,9E+09,9E+09]];
    CONST robtarget rB_v13_t75 := [[1190,40.7072,1893.03],[0.587257,0.193478,0.713218,0.330175],[0,0,4,0],[9E+09,9E+09,9E+09,9E+09,9E+09,9E+09]];
    CONST robtarget rB_v13_t75_c5 := [[1190,40.7072,1893.03],[0.587257,0.193478,0.713218,0.330175],[0,0,0,0],[9E+09,9E+09,9E+09,9E+09,9E+09,9E+09]];
    CONST jointtarget jA_v13_t75 := [[90.0004,48.9364,-7.60278,-44.9996,27.6479,270],[9E+09,9E+09,9E+09,9E+09,9E+09,9E+09]];
    CONST jointtarget jB_v13_t75 := [[0.000224727,-44.6883,35.5904,45.0002,20.1624,360],[9E+09,9E+09,9E+09,9E+09,9E+09,9E+09]];
    CONST jointtarget jBseed_v13_t75 := [[0.000224342,-44.6883,35.5904,45.0002,20.1624,360],[9E+09,9E+09,9E+09,9E+09,9E+09,9E+09]];

    CONST robtarget rA_v13_t83 := [[1209.75,1189.05,1383.72],[0.523784,-0.74058,0.33445,-0.255606],[0,3,-4,0],[9E+09,9E+09,9E+09,9E+09,9E+09,9E+09]];
    CONST robtarget rB_v13_t83 := [[2162.7,0.00705894,2823.41],[0.691878,-0.145976,0.145978,-0.691872],[0,2,-3,0],[9E+09,9E+09,9E+09,9E+09,9E+09,9E+09]];
    CONST robtarget rB_v13_t83_c2 := [[2162.7,0.00705894,2823.41],[0.691878,-0.145976,0.145978,-0.691872],[0,0,-4,0],[9E+09,9E+09,9E+09,9E+09,9E+09,9E+09]];
    CONST jointtarget jA_v13_t83 := [[45.0005,-16.1119,34.8881,270,5.03555,-359.999],[9E+09,9E+09,9E+09,9E+09,9E+09,9E+09]];
    CONST jointtarget jB_v13_t83 := [[0.000194163,37.1843,-75.0804,180,28.276,-270],[9E+09,9E+09,9E+09,9E+09,9E+09,9E+09]];
    CONST jointtarget jBseed_v13_t83 := [[0.000194189,37.1844,-75.0804,180,28.276,-270],[9E+09,9E+09,9E+09,9E+09,9E+09,9E+09]];

    CONST robtarget rA_v13_t87 := [[-541.316,-661.757,3033.67],[0.264237,0.193765,-0.197732,0.92387],[-2,-3,-3,0],[9E+09,9E+09,9E+09,9E+09,9E+09,9E+09]];
    CONST robtarget rB_v13_t87 := [[-0.0206444,-1705.32,-217.381],[0.457066,0.889433,6.08942E-6,-3.74034E-6],[-2,-3,-2,0],[9E+09,9E+09,9E+09,9E+09,9E+09,9E+09]];
    CONST robtarget rB_v13_t87_c4 := [[-0.0206444,-1705.32,-217.381],[0.457066,0.889433,6.08942E-6,-3.74034E-6],[0,-4,0,0],[9E+09,9E+09,9E+09,9E+09,9E+09,9E+09]];
    CONST jointtarget jA_v13_t87 := [[-135.001,-25.3554,-18.1362,-225.001,46.1605,-225.001],[9E+09,9E+09,9E+09,9E+09,9E+09,9E+09]];
    CONST jointtarget jB_v13_t87 := [[-90.0007,49.9802,32.841,-180.001,47.217,-90.0007],[9E+09,9E+09,9E+09,9E+09,9E+09,9E+09]];
    CONST jointtarget jBseed_v13_t87 := [[-90.0007,49.9802,32.841,-180.001,47.217,-90.0007],[9E+09,9E+09,9E+09,9E+09,9E+09,9E+09]];

    CONST robtarget rA_v13_t89 := [[0.00666318,-1887.82,2652.68],[3.47448E-6,1.2188E-7,0.836655,-0.547731],[-1,0,3,0],[9E+09,9E+09,9E+09,9E+09,9E+09,9E+09]];
    CONST robtarget rB_v13_t89 := [[1646.57,1783.86,729.821],[0.228839,-0.923854,0.215229,0.218637],[0,0,2,0],[9E+09,9E+09,9E+09,9E+09,9E+09,9E+09]];
    CONST robtarget rB_v13_t89_c5 := [[1646.57,1783.86,729.821],[0.228839,-0.923854,0.215229,0.218637],[0,0,0,0],[9E+09,9E+09,9E+09,9E+09,9E+09,9E+09]];
    CONST jointtarget jA_v13_t89 := [[-89.9998,8.7985,-38.6001,0.000189978,53.3787,270],[9E+09,9E+09,9E+09,9E+09,9E+09,9E+09]];
    CONST jointtarget jB_v13_t89 := [[44.9991,37.5909,-3.81389,44.9991,55.3288,224.999],[9E+09,9E+09,9E+09,9E+09,9E+09,9E+09]];
    CONST jointtarget jBseed_v13_t89 := [[44.9991,37.5909,-3.8139,44.9991,55.3288,224.999],[9E+09,9E+09,9E+09,9E+09,9E+09,9E+09]];

    CONST robtarget rA_v13_t90 := [[1646.57,1783.86,729.821],[0.228839,-0.923854,0.215229,0.218637],[0,0,2,0],[9E+09,9E+09,9E+09,9E+09,9E+09,9E+09]];
    CONST robtarget rB_v13_t90 := [[382.255,-87.717,3118.13],[0.0853378,-0.00327086,-0.274476,0.957794],[-1,2,3,0],[9E+09,9E+09,9E+09,9E+09,9E+09,9E+09]];
    CONST robtarget rB_v13_t90_c7 := [[382.255,-87.717,3118.13],[0.0853378,-0.00327086,-0.274476,0.957794],[0,-4,4,0],[9E+09,9E+09,9E+09,9E+09,9E+09,9E+09]];
    CONST jointtarget jA_v13_t90 := [[44.9991,37.5909,-3.81389,44.9991,55.3288,224.999],[9E+09,9E+09,9E+09,9E+09,9E+09,9E+09]];
    CONST jointtarget jB_v13_t90 := [[-0.000648657,-34.9394,-20.5246,224.999,47.9696,314.999],[9E+09,9E+09,9E+09,9E+09,9E+09,9E+09]];
    CONST jointtarget jBseed_v13_t90 := [[-0.00064861,-34.9394,-20.5246,224.999,47.9696,314.999],[9E+09,9E+09,9E+09,9E+09,9E+09,9E+09]];

    CONST robtarget rA_v13_t92 := [[2304.74,-0.0059045,2320.74],[0.275742,0.640628,0.265357,0.665693],[-1,-1,1,0],[9E+09,9E+09,9E+09,9E+09,9E+09,9E+09]];
    CONST robtarget rB_v13_t92 := [[50.8216,2521.41,2361.09],[0.853758,-0.353056,0.284217,0.25626],[1,-2,1,0],[9E+09,9E+09,9E+09,9E+09,9E+09,9E+09]];
    CONST robtarget rB_v13_t92_c5 := [[50.8216,2521.41,2361.09],[0.853758,-0.353056,0.284217,0.25626],[0,0,0,0],[9E+09,9E+09,9E+09,9E+09,9E+09,9E+09]];
    CONST jointtarget jA_v13_t92 := [[-0.000144427,19.4299,-34.2082,-0.000149486,12.5797,135],[9E+09,9E+09,9E+09,9E+09,9E+09,9E+09]];
    CONST jointtarget jB_v13_t92 := [[90.0001,37.7264,-57.2986,-135,25.4945,90.0001],[9E+09,9E+09,9E+09,9E+09,9E+09,9E+09]];
    CONST jointtarget jBseed_v13_t92 := [[90.0001,37.7264,-57.2985,-135,25.4946,90.0001],[9E+09,9E+09,9E+09,9E+09,9E+09,9E+09]];

    CONST robtarget rA_v13_t96 := [[-12.6098,-1883.18,1114.14],[0.222193,0.313192,-0.805579,0.451201],[-2,-2,-1,0],[9E+09,9E+09,9E+09,9E+09,9E+09,9E+09]];
    CONST robtarget rB_v13_t96 := [[5.74273,-2118.55,2681.51],[0.797399,0.466576,0.209201,-0.320463],[-2,1,2,0],[9E+09,9E+09,9E+09,9E+09,9E+09,9E+09]];
    CONST robtarget rB_v13_t96_c4 := [[5.74273,-2118.55,2681.51],[0.797399,0.466576,0.209201,-0.320463],[0,-4,0,0],[9E+09,9E+09,9E+09,9E+09,9E+09,9E+09]];
    CONST robtarget rB_v13_t96_c5 := [[5.74273,-2118.55,2681.51],[0.797399,0.466576,0.209201,-0.320463],[0,0,0,0],[9E+09,9E+09,9E+09,9E+09,9E+09,9E+09]];
    CONST jointtarget jA_v13_t96 := [[-90.0008,-1.2653,30.9684,-90.0008,4.32142,-45.0008],[9E+09,9E+09,9E+09,9E+09,9E+09,9E+09]];
    CONST jointtarget jB_v13_t96 := [[-90.001,18.5693,-45.0987,134.999,2.80526,269.999],[9E+09,9E+09,9E+09,9E+09,9E+09,9E+09]];
    CONST jointtarget jBseed_v13_t96 := [[-90.001,18.5693,-45.0987,134.999,2.80526,269.999],[9E+09,9E+09,9E+09,9E+09,9E+09,9E+09]];

    CONST robtarget rA_v13_t97 := [[5.74273,-2118.55,2681.51],[0.797399,0.466576,0.209201,-0.320463],[-2,1,2,0],[9E+09,9E+09,9E+09,9E+09,9E+09,9E+09]];
    CONST robtarget rB_v13_t97 := [[2174,-2043.97,1243.12],[0.214617,-0.641013,0.370961,-0.636734],[-1,-3,1,0],[9E+09,9E+09,9E+09,9E+09,9E+09,9E+09]];
    CONST robtarget rB_v13_t97_c5 := [[2174,-2043.97,1243.12],[0.214617,-0.641013,0.370961,-0.636734],[0,0,0,0],[9E+09,9E+09,9E+09,9E+09,9E+09,9E+09]];
    CONST jointtarget jA_v13_t97 := [[-90.001,18.5693,-45.0987,134.999,2.80526,269.999],[9E+09,9E+09,9E+09,9E+09,9E+09,9E+09]];
    CONST jointtarget jB_v13_t97 := [[-44.9993,59.3774,-52.7043,-269.999,33.3885,135.001],[9E+09,9E+09,9E+09,9E+09,9E+09,9E+09]];
    CONST jointtarget jBseed_v13_t97 := [[-44.9993,59.3774,-52.7042,-269.999,33.3885,135.001],[9E+09,9E+09,9E+09,9E+09,9E+09,9E+09]];

    CONST robtarget rA_v13_t100 := [[-354.926,363.102,3184.79],[0.681855,-0.281449,0.0166212,0.67497],[1,-1,0,0],[9E+09,9E+09,9E+09,9E+09,9E+09,9E+09]];
    CONST robtarget rB_v13_t100 := [[53.8414,916.112,3075.79],[0.406599,7.66207E-5,0.396356,0.823152],[1,-1,1,0],[9E+09,9E+09,9E+09,9E+09,9E+09,9E+09]];
    CONST robtarget rB_v13_t100_c2 := [[53.8414,916.112,3075.79],[0.406599,7.66207E-5,0.396356,0.823152],[0,0,-4,0],[9E+09,9E+09,9E+09,9E+09,9E+09,9E+09]];
    CONST robtarget rB_v13_t100_c5 := [[53.8414,916.112,3075.79],[0.406599,7.66207E-5,0.396356,0.823152],[0,0,0,0],[9E+09,9E+09,9E+09,9E+09,9E+09,9E+09]];
    CONST jointtarget jA_v13_t100 := [[135,-30.5997,-26.7019,-89.9996,1.98492,45.0002],[9E+09,9E+09,9E+09,9E+09,9E+09,9E+09]];
    CONST jointtarget jB_v13_t100 := [[90.0005,-22.8321,-23.5954,-89.9995,18.811,135],[9E+09,9E+09,9E+09,9E+09,9E+09,9E+09]];
    CONST jointtarget jBseed_v13_t100 := [[90.0005,-22.8321,-23.5954,-89.9995,18.811,135],[9E+09,9E+09,9E+09,9E+09,9E+09,9E+09]];

    CONST robtarget rA_v13_t101 := [[53.8414,916.112,3075.79],[0.406599,7.66207E-5,0.396356,0.823152],[1,-1,1,0],[9E+09,9E+09,9E+09,9E+09,9E+09,9E+09]];
    CONST robtarget rB_v13_t101 := [[1416.88,1593.11,2695.45],[0.490653,-0.282732,-0.501204,-0.654306],[0,1,1,0],[9E+09,9E+09,9E+09,9E+09,9E+09,9E+09]];
    CONST robtarget rB_v13_t101_c4 := [[1416.88,1593.11,2695.45],[0.490653,-0.282732,-0.501204,-0.654306],[0,-4,0,0],[9E+09,9E+09,9E+09,9E+09,9E+09,9E+09]];
    CONST robtarget rB_v13_t101_c5 := [[1416.88,1593.11,2695.45],[0.490653,-0.282732,-0.501204,-0.654306],[0,0,0,0],[9E+09,9E+09,9E+09,9E+09,9E+09,9E+09]];
    CONST jointtarget jA_v13_t101 := [[90.0005,-22.8321,-23.5954,-89.9995,18.811,135],[9E+09,9E+09,9E+09,9E+09,9E+09,9E+09]];
    CONST jointtarget jB_v13_t101 := [[45.0003,25.3957,-55.8742,90.0003,48.2553,90.0003],[9E+09,9E+09,9E+09,9E+09,9E+09,9E+09]];
    CONST jointtarget jBseed_v13_t101 := [[45.0003,25.3957,-55.8742,90.0003,48.2553,90.0003],[9E+09,9E+09,9E+09,9E+09,9E+09,9E+09]];

    CONST robtarget rA_v13_t102 := [[1416.88,1593.11,2695.45],[0.490653,-0.282732,-0.501204,-0.654306],[0,1,1,0],[9E+09,9E+09,9E+09,9E+09,9E+09,9E+09]];
    CONST robtarget rB_v13_t102 := [[314.295,-314.297,3349.86],[0.984597,-0.123632,-0.123631,-5.87079E-6],[-1,1,-2,0],[9E+09,9E+09,9E+09,9E+09,9E+09,9E+09]];
    CONST robtarget rB_v13_t102_c4 := [[314.295,-314.297,3349.86],[0.984597,-0.123632,-0.123631,-5.87079E-6],[0,-4,0,0],[9E+09,9E+09,9E+09,9E+09,9E+09,9E+09]];
    CONST robtarget rB_v13_t102_c5 := [[314.295,-314.297,3349.86],[0.984597,-0.123632,-0.123631,-5.87079E-6],[0,0,0,0],[9E+09,9E+09,9E+09,9E+09,9E+09,9E+09]];
    CONST jointtarget jA_v13_t102 := [[45.0003,25.3957,-55.8742,90.0003,48.2553,90.0003],[9E+09,9E+09,9E+09,9E+09,9E+09,9E+09]];
    CONST jointtarget jB_v13_t102 := [[-45.0002,-18.8037,-43.4681,180,47.8671,-135],[9E+09,9E+09,9E+09,9E+09,9E+09,9E+09]];
    CONST jointtarget jBseed_v13_t102 := [[-45.0002,-18.8037,-43.4681,180,47.8671,-135],[9E+09,9E+09,9E+09,9E+09,9E+09,9E+09]];

    CONST robtarget rA_v13_t107 := [[2431.71,-0.0390227,843.612],[0.187944,0.804795,0.333365,0.453707],[-1,1,-1,0],[9E+09,9E+09,9E+09,9E+09,9E+09,9E+09]];
    CONST robtarget rB_v13_t107 := [[75.8357,-496.85,3138.18],[0.968398,0.0619882,0.229655,0.0749749],[-1,1,3,0],[9E+09,9E+09,9E+09,9E+09,9E+09,9E+09]];
    CONST robtarget rB_v13_t107_c5 := [[75.8357,-496.85,3138.18],[0.968398,0.0619882,0.229655,0.0749749],[0,0,0,0],[9E+09,9E+09,9E+09,9E+09,9E+09,9E+09]];
    CONST robtarget rB_v13_t107_c8 := [[75.8357,-496.85,3138.18],[0.968398,0.0619882,0.229655,0.0749749],[0,0,4,0],[9E+09,9E+09,9E+09,9E+09,9E+09,9E+09]];
    CONST jointtarget jA_v13_t107 := [[-0.000922588,30.8817,3.18461,179.999,2.89133,-45.0009],[9E+09,9E+09,9E+09,9E+09,9E+09,9E+09]];
    CONST jointtarget jB_v13_t107 := [[-89.9997,-31.7276,-22.1156,135,39.9548,315],[9E+09,9E+09,9E+09,9E+09,9E+09,9E+09]];
    CONST jointtarget jBseed_v13_t107 := [[-89.9997,-31.7277,-22.1155,135,39.9548,315],[9E+09,9E+09,9E+09,9E+09,9E+09,9E+09]];

    CONST robtarget rA_v13_t111 := [[96.8943,-2752.79,628.587],[0.280014,-0.169824,0.927638,-0.179553],[-2,0,-2,0],[9E+09,9E+09,9E+09,9E+09,9E+09,9E+09]];
    CONST robtarget rB_v13_t111 := [[2318.08,-0.0277569,744.221],[8.12678E-6,0.870399,5.59839E-6,0.492346],[-1,-3,-1,0],[9E+09,9E+09,9E+09,9E+09,9E+09,9E+09]];
    CONST robtarget rB_v13_t111_c2 := [[2318.08,-0.0277569,744.221],[8.12678E-6,0.870399,5.59839E-6,0.492346],[0,0,-4,0],[9E+09,9E+09,9E+09,9E+09,9E+09,9E+09]];
    CONST robtarget rB_v13_t111_c5 := [[2318.08,-0.0277569,744.221],[8.12678E-6,0.870399,5.59839E-6,0.492346],[0,0,0,0],[9E+09,9E+09,9E+09,9E+09,9E+09,9E+09]];
    CONST jointtarget jA_v13_t111 := [[-90.001,55.9825,-28.4515,44.999,55.1805,-135.001],[9E+09,9E+09,9E+09,9E+09,9E+09,9E+09]];
    CONST jointtarget jB_v13_t111 := [[-0.000693228,28.3035,11.0163,-180.001,8.30958,-0.000693228],[9E+09,9E+09,9E+09,9E+09,9E+09,9E+09]];
    CONST jointtarget jBseed_v13_t111 := [[-0.000693228,28.3035,11.0163,-180.001,8.30958,-0.000693228],[9E+09,9E+09,9E+09,9E+09,9E+09,9E+09]];

    CONST robtarget rA_v13_t112 := [[2318.08,-0.0277569,744.221],[8.12678E-6,0.870399,5.59839E-6,0.492346],[-1,-3,-1,0],[9E+09,9E+09,9E+09,9E+09,9E+09,9E+09]];
    CONST robtarget rB_v13_t112 := [[2007.44,2007.37,1915.74],[0.957431,-0.20412,0.204109,-2.05703E-5],[0,1,-3,0],[9E+09,9E+09,9E+09,9E+09,9E+09,9E+09]];
    CONST robtarget rB_v13_t112_c1 := [[2007.44,2007.37,1915.74],[0.957431,-0.20412,0.204109,-2.05703E-5],[0,-4,-4,0],[9E+09,9E+09,9E+09,9E+09,9E+09,9E+09]];
    CONST robtarget rB_v13_t112_c4 := [[2007.44,2007.37,1915.74],[0.957431,-0.20412,0.204109,-2.05703E-5],[0,-4,0,0],[9E+09,9E+09,9E+09,9E+09,9E+09,9E+09]];
    CONST jointtarget jA_v13_t112 := [[-0.000693228,28.3035,11.0163,-180.001,8.30958,-0.000693228],[9E+09,9E+09,9E+09,9E+09,9E+09,9E+09]];
    CONST jointtarget jB_v13_t112 := [[44.999,58.7219,-71.0218,179.999,44.1444,-225.001],[9E+09,9E+09,9E+09,9E+09,9E+09,9E+09]];
    CONST jointtarget jBseed_v13_t112 := [[44.999,58.7219,-71.0218,179.999,44.1444,-225.001],[9E+09,9E+09,9E+09,9E+09,9E+09,9E+09]];

    CONST robtarget rA_v13_t113 := [[2007.44,2007.37,1915.74],[0.957431,-0.20412,0.204109,-2.05703E-5],[0,1,-3,0],[9E+09,9E+09,9E+09,9E+09,9E+09,9E+09]];
    CONST robtarget rB_v13_t113 := [[0.0193565,2208.4,1461.66],[0.51111,-0.488629,-0.488634,-0.511121],[0,1,3,0],[9E+09,9E+09,9E+09,9E+09,9E+09,9E+09]];
    CONST robtarget rB_v13_t113_c2 := [[0.0193565,2208.4,1461.66],[0.51111,-0.488629,-0.488634,-0.511121],[0,0,-4,0],[9E+09,9E+09,9E+09,9E+09,9E+09,9E+09]];
    CONST robtarget rB_v13_t113_c5 := [[0.0193565,2208.4,1461.66],[0.51111,-0.488629,-0.488634,-0.511121],[0,0,0,0],[9E+09,9E+09,9E+09,9E+09,9E+09,9E+09]];
    CONST jointtarget jA_v13_t113 := [[44.999,58.7219,-71.0218,179.999,44.1444,-225.001],[9E+09,9E+09,9E+09,9E+09,9E+09,9E+09]];
    CONST jointtarget jB_v13_t113 := [[89.9995,9.98138,9.17539,179.999,21.7334,359.999],[9E+09,9E+09,9E+09,9E+09,9E+09,9E+09]];
    CONST jointtarget jBseed_v13_t113 := [[89.9995,9.98138,9.17538,179.999,21.7335,359.999],[9E+09,9E+09,9E+09,9E+09,9E+09,9E+09]];

    CONST robtarget rA_v13_t117 := [[1214.62,1332.39,2894.13],[0.215949,-0.0386439,0.503445,0.835713],[0,-4,3,0],[9E+09,9E+09,9E+09,9E+09,9E+09,9E+09]];
    CONST robtarget rB_v13_t117 := [[2050.22,30.7295,1041.48],[0.137064,0.746719,0.357299,0.544024],[-1,-3,-1,0],[9E+09,9E+09,9E+09,9E+09,9E+09,9E+09]];
    CONST robtarget rB_v13_t117_c7 := [[2050.22,30.7295,1041.48],[0.137064,0.746719,0.357299,0.544024],[0,-4,4,0],[9E+09,9E+09,9E+09,9E+09,9E+09,9E+09]];
    CONST jointtarget jA_v13_t117 := [[44.9994,10.2011,-44.6345,-270.001,29.9167,359.999],[9E+09,9E+09,9E+09,9E+09,9E+09,9E+09]];
    CONST jointtarget jB_v13_t117 := [[-0.000269411,8.76553,24.1722,-225,15.0884,-0.000273979],[9E+09,9E+09,9E+09,9E+09,9E+09,9E+09]];
    CONST jointtarget jBseed_v13_t117 := [[-0.000269265,8.76553,24.1722,-225,15.0884,-0.000269265],[9E+09,9E+09,9E+09,9E+09,9E+09,9E+09]];

    CONST robtarget rA_v13_t118 := [[2050.22,30.7295,1041.48],[0.137064,0.746719,0.357299,0.544024],[-1,-3,-1,0],[9E+09,9E+09,9E+09,9E+09,9E+09,9E+09]];
    CONST robtarget rB_v13_t118 := [[770.944,-631.778,3167.1],[0.247142,0.130747,0.282449,0.917632],[-1,-3,-4,0],[9E+09,9E+09,9E+09,9E+09,9E+09,9E+09]];
    CONST robtarget rB_v13_t118_c4 := [[770.944,-631.778,3167.1],[0.247142,0.130747,0.282449,0.917632],[0,-4,0,0],[9E+09,9E+09,9E+09,9E+09,9E+09,9E+09]];
    CONST jointtarget jA_v13_t118 := [[-0.000269411,8.76553,24.1722,-225,15.0884,-0.000273979],[9E+09,9E+09,9E+09,9E+09,9E+09,9E+09]];
    CONST jointtarget jB_v13_t118 := [[-44.9999,-11.8931,-35.0017,-225,56.4403,-315],[9E+09,9E+09,9E+09,9E+09,9E+09,9E+09]];
    CONST jointtarget jBseed_v13_t118 := [[-44.9999,-11.8931,-35.0017,-225,56.4403,-315],[9E+09,9E+09,9E+09,9E+09,9E+09,9E+09]];

    CONST robtarget rA_v13_t119 := [[770.944,-631.778,3167.1],[0.247142,0.130747,0.282449,0.917632],[-1,-3,-4,0],[9E+09,9E+09,9E+09,9E+09,9E+09,9E+09]];
    CONST robtarget rB_v13_t119 := [[585.376,-524.146,3452.61],[0.705957,-0.128464,0.185296,-0.671407],[-1,0,2,0],[9E+09,9E+09,9E+09,9E+09,9E+09,9E+09]];
    CONST robtarget rB_v13_t119_c1 := [[585.376,-524.146,3452.61],[0.705957,-0.128464,0.185296,-0.671407],[0,-4,-4,0],[9E+09,9E+09,9E+09,9E+09,9E+09,9E+09]];
    CONST jointtarget jA_v13_t119 := [[-44.9999,-11.8931,-35.0017,-225,56.4403,-315],[9E+09,9E+09,9E+09,9E+09,9E+09,9E+09]];
    CONST jointtarget jB_v13_t119 := [[-45.0004,1.18104,-69.6371,89.9997,15.0279,225],[9E+09,9E+09,9E+09,9E+09,9E+09,9E+09]];
    CONST jointtarget jBseed_v13_t119 := [[-45.0004,1.18106,-69.6371,89.9996,15.0279,225],[9E+09,9E+09,9E+09,9E+09,9E+09,9E+09]];

    CONST robtarget rA_v13_t120 := [[585.376,-524.146,3452.61],[0.705957,-0.128464,0.185296,-0.671407],[-1,0,2,0],[9E+09,9E+09,9E+09,9E+09,9E+09,9E+09]];
    CONST robtarget rB_v13_t120 := [[745.276,-889.135,3139.17],[0.113201,0.198173,-0.667598,0.708678],[-1,-1,-2,0],[9E+09,9E+09,9E+09,9E+09,9E+09,9E+09]];
    CONST robtarget rB_v13_t120_c8 := [[745.276,-889.135,3139.17],[0.113201,0.198173,-0.667598,0.708678],[0,0,4,0],[9E+09,9E+09,9E+09,9E+09,9E+09,9E+09]];
    CONST jointtarget jA_v13_t120 := [[-45.0004,1.18104,-69.6371,89.9997,15.0279,225],[9E+09,9E+09,9E+09,9E+09,9E+09,9E+09]];
    CONST jointtarget jB_v13_t120 := [[-45.0005,-4.2903,-48.0505,-45.0005,59.4671,-90.0005],[9E+09,9E+09,9E+09,9E+09,9E+09,9E+09]];
    CONST jointtarget jBseed_v13_t120 := [[-45.0005,-4.29029,-48.0505,-45.0005,59.4671,-90.0005],[9E+09,9E+09,9E+09,9E+09,9E+09,9E+09]];

    CONST robtarget rA_v13_t123 := [[-37.6454,-1260.86,3135.01],[0.952539,0.282193,-0.105016,-0.0448104],[-2,-2,2,0],[9E+09,9E+09,9E+09,9E+09,9E+09,9E+09]];
    CONST robtarget rB_v13_t123 := [[2179.41,98.2912,2547.62],[0.795588,-0.440221,0.390919,-0.142923],[-1,-4,-2,0],[9E+09,9E+09,9E+09,9E+09,9E+09,9E+09]];
    CONST robtarget rB_v13_t123_c4 := [[2179.41,98.2912,2547.62],[0.795588,-0.440221,0.390919,-0.142923],[0,-4,0,0],[9E+09,9E+09,9E+09,9E+09,9E+09,9E+09]];
    CONST robtarget rB_v13_t123_c5 := [[2179.41,98.2912,2547.62],[0.795588,-0.440221,0.390919,-0.142923],[0,0,0,0],[9E+09,9E+09,9E+09,9E+09,9E+09,9E+09]];
    CONST jointtarget jA_v13_t123 := [[-90.0006,-6.45466,-37.3425,-135.001,18.5839,224.999],[9E+09,9E+09,9E+09,9E+09,9E+09,9E+09]];
    CONST jointtarget jB_v13_t123 := [[-0.000731288,19.7632,-42.0676,-270.001,36.0674,-135.001],[9E+09,9E+09,9E+09,9E+09,9E+09,9E+09]];
    CONST jointtarget jBseed_v13_t123 := [[-0.000731376,19.7632,-42.0676,-270.001,36.0674,-135.001],[9E+09,9E+09,9E+09,9E+09,9E+09,9E+09]];

    CONST robtarget rA_v13_t125 := [[2407.3,77.537,1250.14],[0.198137,-0.805007,-0.133637,-0.542997],[0,1,1,0],[9E+09,9E+09,9E+09,9E+09,9E+09,9E+09]];
    CONST robtarget rB_v13_t125 := [[1405.79,1525.14,617.056],[0.359597,-0.702269,0.564369,0.24289],[0,1,-2,0],[9E+09,9E+09,9E+09,9E+09,9E+09,9E+09]];
    CONST robtarget rB_v13_t125_c5 := [[1405.79,1525.14,617.056],[0.359597,-0.702269,0.564369,0.24289],[0,0,0,0],[9E+09,9E+09,9E+09,9E+09,9E+09,9E+09]];
    CONST robtarget rB_v13_t125_c8 := [[1405.79,1525.14,617.056],[0.359597,-0.702269,0.564369,0.24289],[0,0,4,0],[9E+09,9E+09,9E+09,9E+09,9E+09,9E+09]];
    CONST jointtarget jA_v13_t125 := [[0.00067944,23.1544,-1.15573,90.0007,27.6534,90.0007],[9E+09,9E+09,9E+09,9E+09,9E+09,9E+09]];
    CONST jointtarget jB_v13_t125 := [[45.0008,23.0335,23.216,90.0008,30.3452,-134.999],[9E+09,9E+09,9E+09,9E+09,9E+09,9E+09]];
    CONST jointtarget jBseed_v13_t125 := [[45.0008,23.0335,23.216,90.0008,30.3452,-134.999],[9E+09,9E+09,9E+09,9E+09,9E+09,9E+09]];

    CONST robtarget rA_v13_t126 := [[1405.79,1525.14,617.056],[0.359597,-0.702269,0.564369,0.24289],[0,1,-2,0],[9E+09,9E+09,9E+09,9E+09,9E+09,9E+09]];
    CONST robtarget rB_v13_t126 := [[-1845.63,1845.64,2203.8],[2.8721E-6,-0.147011,0.14701,0.978149],[1,-3,-2,0],[9E+09,9E+09,9E+09,9E+09,9E+09,9E+09]];
    CONST robtarget rB_v13_t126_c2 := [[-1845.63,1845.64,2203.8],[2.8721E-6,-0.147011,0.14701,0.978149],[0,0,-4,0],[9E+09,9E+09,9E+09,9E+09,9E+09,9E+09]];
    CONST jointtarget jA_v13_t126 := [[45.0008,23.0335,23.216,90.0008,30.3452,-134.999],[9E+09,9E+09,9E+09,9E+09,9E+09,9E+09]];
    CONST jointtarget jB_v13_t126 := [[135,43.3039,-57.2152,-180,52.0896,-135],[9E+09,9E+09,9E+09,9E+09,9E+09,9E+09]];
    CONST jointtarget jBseed_v13_t126 := [[135,43.3039,-57.2152,-180,52.0896,-135],[9E+09,9E+09,9E+09,9E+09,9E+09,9E+09]];

    CONST robtarget rA_v13_t127 := [[-1845.63,1845.64,2203.8],[2.8721E-6,-0.147011,0.14701,0.978149],[1,-3,-2,0],[9E+09,9E+09,9E+09,9E+09,9E+09,9E+09]];
    CONST robtarget rB_v13_t127 := [[410.531,0.00543862,2588.65],[0.827972,-0.169789,0.409911,-0.342939],[0,0,-1,0],[9E+09,9E+09,9E+09,9E+09,9E+09,9E+09]];
    CONST robtarget rB_v13_t127_c5 := [[410.531,0.00543862,2588.65],[0.827972,-0.169789,0.409911,-0.342939],[0,0,0,0],[9E+09,9E+09,9E+09,9E+09,9E+09,9E+09]];
    CONST jointtarget jA_v13_t127 := [[135,43.3039,-57.2152,-180,52.0896,-135],[9E+09,9E+09,9E+09,9E+09,9E+09,9E+09]];
    CONST jointtarget jB_v13_t127 := [[0.000713353,-59.8865,13.6784,0.000727059,8.88638,-44.9993],[9E+09,9E+09,9E+09,9E+09,9E+09,9E+09]];
    CONST jointtarget jBseed_v13_t127 := [[0.000714164,-59.8865,13.6784,0.000714164,8.88638,-44.9993],[9E+09,9E+09,9E+09,9E+09,9E+09,9E+09]];

    CONST robtarget rA_v13_t128 := [[410.531,0.00543862,2588.65],[0.827972,-0.169789,0.409911,-0.342939],[0,0,-1,0],[9E+09,9E+09,9E+09,9E+09,9E+09,9E+09]];
    CONST robtarget rB_v13_t128 := [[-62.8394,316.019,3100.29],[0.651426,-0.193118,-0.0723435,0.730148],[1,1,-2,0],[9E+09,9E+09,9E+09,9E+09,9E+09,9E+09]];
    CONST robtarget rB_v13_t128_c4 := [[-62.8394,316.019,3100.29],[0.651426,-0.193118,-0.0723435,0.730148],[0,-4,0,0],[9E+09,9E+09,9E+09,9E+09,9E+09,9E+09]];
    CONST robtarget rB_v13_t128_c5 := [[-62.8394,316.019,3100.29],[0.651426,-0.193118,-0.0723435,0.730148],[0,0,0,0],[9E+09,9E+09,9E+09,9E+09,9E+09,9E+09]];
    CONST jointtarget jA_v13_t128 := [[0.000713353,-59.8865,13.6784,0.000727059,8.88638,-44.9993],[9E+09,9E+09,9E+09,9E+09,9E+09,9E+09]];
    CONST jointtarget jB_v13_t128 := [[90.0007,-38.9496,-18.0251,135.001,32.1488,-134.999],[9E+09,9E+09,9E+09,9E+09,9E+09,9E+09]];
    CONST jointtarget jBseed_v13_t128 := [[90.0007,-38.9496,-18.0251,135.001,32.1488,-134.999],[9E+09,9E+09,9E+09,9E+09,9E+09,9E+09]];

    CONST robtarget rA_v13_t129 := [[-62.8394,316.019,3100.29],[0.651426,-0.193118,-0.0723435,0.730148],[1,1,-2,0],[9E+09,9E+09,9E+09,9E+09,9E+09,9E+09]];
    CONST robtarget rB_v13_t129 := [[1765.43,-22.7857,1045.07],[0.518959,0.352129,0.764353,0.149836],[-1,-2,-3,0],[9E+09,9E+09,9E+09,9E+09,9E+09,9E+09]];
    CONST robtarget rB_v13_t129_c2 := [[1765.43,-22.7857,1045.07],[0.518959,0.352129,0.764353,0.149836],[0,0,-4,0],[9E+09,9E+09,9E+09,9E+09,9E+09,9E+09]];
    CONST jointtarget jA_v13_t129 := [[90.0007,-38.9496,-18.0251,135.001,32.1488,-134.999],[9E+09,9E+09,9E+09,9E+09,9E+09,9E+09]];
    CONST jointtarget jB_v13_t129 := [[-9.49629E-5,-5.84674,38.6215,-135,11.124,-180],[9E+09,9E+09,9E+09,9E+09,9E+09,9E+09]];
    CONST jointtarget jBseed_v13_t129 := [[-9.49431E-5,-5.84674,38.6215,-135,11.124,-180],[9E+09,9E+09,9E+09,9E+09,9E+09,9E+09]];

    CONST robtarget rA_v13_t130 := [[1765.43,-22.7857,1045.07],[0.518959,0.352129,0.764353,0.149836],[-1,-2,-3,0],[9E+09,9E+09,9E+09,9E+09,9E+09,9E+09]];
    CONST robtarget rB_v13_t130 := [[1100.39,-1154.71,1544.68],[0.185197,-0.200898,0.674512,-0.685839],[-1,2,-4,0],[9E+09,9E+09,9E+09,9E+09,9E+09,9E+09]];
    CONST robtarget rB_v13_t130_c2 := [[1100.39,-1154.71,1544.68],[0.185197,-0.200898,0.674512,-0.685839],[0,0,-4,0],[9E+09,9E+09,9E+09,9E+09,9E+09,9E+09]];
    CONST robtarget rB_v13_t130_c5 := [[1100.39,-1154.71,1544.68],[0.185197,-0.200898,0.674512,-0.685839],[0,0,0,0],[9E+09,9E+09,9E+09,9E+09,9E+09,9E+09]];
    CONST jointtarget jA_v13_t130 := [[-9.49629E-5,-5.84674,38.6215,-135,11.124,-180],[9E+09,9E+09,9E+09,9E+09,9E+09,9E+09]];
    CONST jointtarget jB_v13_t130 := [[-44.9994,-23.1544,36.2807,225.001,18.9904,-314.999],[9E+09,9E+09,9E+09,9E+09,9E+09,9E+09]];
    CONST jointtarget jBseed_v13_t130 := [[-44.9994,-23.1544,36.2807,225.001,18.9904,-314.999],[9E+09,9E+09,9E+09,9E+09,9E+09,9E+09]];

    CONST robtarget rA_v13_t131 := [[1100.39,-1154.71,1544.68],[0.185197,-0.200898,0.674512,-0.685839],[-1,2,-4,0],[9E+09,9E+09,9E+09,9E+09,9E+09,9E+09]];
    CONST robtarget rB_v13_t131 := [[-48.5548,-2118,2755.18],[0.0721428,-0.128098,-0.485437,0.861822],[-1,-1,0,0],[9E+09,9E+09,9E+09,9E+09,9E+09,9E+09]];
    CONST robtarget rB_v13_t131_c3 := [[-48.5548,-2118,2755.18],[0.0721428,-0.128098,-0.485437,0.861822],[0,4,-4,0],[9E+09,9E+09,9E+09,9E+09,9E+09,9E+09]];
    CONST jointtarget jA_v13_t131 := [[-44.9994,-23.1544,36.2807,225.001,18.9904,-314.999],[9E+09,9E+09,9E+09,9E+09,9E+09,9E+09]];
    CONST jointtarget jB_v13_t131 := [[-89.9996,23.2203,-54.438,-89.9996,16.9085,0.000444281],[9E+09,9E+09,9E+09,9E+09,9E+09,9E+09]];
    CONST jointtarget jBseed_v13_t131 := [[-89.9996,23.2203,-54.438,-89.9996,16.9085,0.000432661],[9E+09,9E+09,9E+09,9E+09,9E+09,9E+09]];

    CONST robtarget rA_v13_t132 := [[-48.5548,-2118,2755.18],[0.0721428,-0.128098,-0.485437,0.861822],[-1,-1,0,0],[9E+09,9E+09,9E+09,9E+09,9E+09,9E+09]];
    CONST robtarget rB_v13_t132 := [[1390.94,1390.9,1050.94],[0.518524,-0.316736,0.764648,0.214766],[0,-3,-3,0],[9E+09,9E+09,9E+09,9E+09,9E+09,9E+09]];
    CONST robtarget rB_v13_t132_c1 := [[1390.94,1390.9,1050.94],[0.518524,-0.316736,0.764648,0.214766],[0,-4,-4,0],[9E+09,9E+09,9E+09,9E+09,9E+09,9E+09]];
    CONST robtarget rB_v13_t132_c4 := [[1390.94,1390.9,1050.94],[0.518524,-0.316736,0.764648,0.214766],[0,-4,0,0],[9E+09,9E+09,9E+09,9E+09,9E+09,9E+09]];
    CONST jointtarget jA_v13_t132 := [[-89.9996,23.2203,-54.438,-89.9996,16.9085,0.000444281],[9E+09,9E+09,9E+09,9E+09,9E+09,9E+09]];
    CONST jointtarget jB_v13_t132 := [[44.9991,4.33424,28.6236,-180.001,11.2412,-180.001],[9E+09,9E+09,9E+09,9E+09,9E+09,9E+09]];
    CONST jointtarget jBseed_v13_t132 := [[44.9991,4.33424,28.6236,-180.001,11.2412,-180.001],[9E+09,9E+09,9E+09,9E+09,9E+09,9E+09]];

    CONST robtarget rA_v13_t133 := [[1390.94,1390.9,1050.94],[0.518524,-0.316736,0.764648,0.214766],[0,-3,-3,0],[9E+09,9E+09,9E+09,9E+09,9E+09,9E+09]];
    CONST robtarget rB_v13_t133 := [[1342.08,-1183.48,1344.27],[0.159264,0.772436,0.201875,0.58071],[-1,0,0,0],[9E+09,9E+09,9E+09,9E+09,9E+09,9E+09]];
    CONST robtarget rB_v13_t133_c4 := [[1342.08,-1183.48,1344.27],[0.159264,0.772436,0.201875,0.58071],[0,-4,0,0],[9E+09,9E+09,9E+09,9E+09,9E+09,9E+09]];
    CONST jointtarget jA_v13_t133 := [[44.9991,4.33424,28.6236,-180.001,11.2412,-180.001],[9E+09,9E+09,9E+09,9E+09,9E+09,9E+09]];
    CONST jointtarget jB_v13_t133 := [[-45.0005,-8.23084,30.0043,89.9995,42.1943,44.9995],[9E+09,9E+09,9E+09,9E+09,9E+09,9E+09]];
    CONST jointtarget jBseed_v13_t133 := [[-45.0005,-8.23084,30.0043,89.9995,42.1943,44.9995],[9E+09,9E+09,9E+09,9E+09,9E+09,9E+09]];

    CONST robtarget rA_v13_t135 := [[-1261.78,1402.21,2455.87],[0.48658,-0.265535,-0.279459,-0.783985],[1,2,3,0],[9E+09,9E+09,9E+09,9E+09,9E+09,9E+09]];
    CONST robtarget rB_v13_t135 := [[-1906.93,1805.39,537.235],[0.574225,0.0960478,-0.762112,-0.283242],[1,1,3,0],[9E+09,9E+09,9E+09,9E+09,9E+09,9E+09]];
    CONST robtarget rB_v13_t135_c8 := [[-1906.93,1805.39,537.235],[0.574225,0.0960478,-0.762112,-0.283242],[0,0,4,0],[9E+09,9E+09,9E+09,9E+09,9E+09,9E+09]];
    CONST jointtarget jA_v13_t135 := [[135,1.94281,-15.1845,225,57.2442,270],[9E+09,9E+09,9E+09,9E+09,9E+09,9E+09]];
    CONST jointtarget jB_v13_t135 := [[134.999,48.7936,-8.83664,134.999,37.4627,359.999],[9E+09,9E+09,9E+09,9E+09,9E+09,9E+09]];
    CONST jointtarget jBseed_v13_t135 := [[134.999,48.7936,-8.83664,134.999,37.4627,359.999],[9E+09,9E+09,9E+09,9E+09,9E+09,9E+09]];

    CONST robtarget rA_v13_t143 := [[911.303,937.148,1685.7],[0.0393846,-0.451772,-0.505845,-0.733806],[0,1,3,0],[9E+09,9E+09,9E+09,9E+09,9E+09,9E+09]];
    CONST robtarget rB_v13_t143 := [[-1117.5,1117.52,3101.47],[0.382565,0.00916495,-0.0221194,-0.923618],[1,-3,-2,0],[9E+09,9E+09,9E+09,9E+09,9E+09,9E+09]];
    CONST robtarget rB_v13_t143_c8 := [[-1117.5,1117.52,3101.47],[0.382565,0.00916495,-0.0221194,-0.923618],[0,0,4,0],[9E+09,9E+09,9E+09,9E+09,9E+09,9E+09]];
    CONST jointtarget jA_v13_t143 := [[44.9998,-40.755,42.458,135,8.90469,360],[9E+09,9E+09,9E+09,9E+09,9E+09,9E+09]];
    CONST jointtarget jB_v13_t143 := [[135,11.0617,-52.0219,-180,46.296,-90.0004],[9E+09,9E+09,9E+09,9E+09,9E+09,9E+09]];
    CONST jointtarget jBseed_v13_t143 := [[135,11.0617,-52.0219,-180,46.296,-90.0004],[9E+09,9E+09,9E+09,9E+09,9E+09,9E+09]];

    CONST robtarget rA_v13_t144 := [[-1117.5,1117.52,3101.47],[0.382565,0.00916495,-0.0221194,-0.923618],[1,-3,-2,0],[9E+09,9E+09,9E+09,9E+09,9E+09,9E+09]];
    CONST robtarget rB_v13_t144 := [[983.46,1103.96,351.653],[0.159979,-0.959864,-0.0681744,0.220047],[0,0,-2,0],[9E+09,9E+09,9E+09,9E+09,9E+09,9E+09]];
    CONST robtarget rB_v13_t144_c2 := [[983.46,1103.96,351.653],[0.159979,-0.959864,-0.0681744,0.220047],[0,0,-4,0],[9E+09,9E+09,9E+09,9E+09,9E+09,9E+09]];
    CONST jointtarget jA_v13_t144 := [[135,11.0617,-52.0219,-180,46.296,-90.0004],[9E+09,9E+09,9E+09,9E+09,9E+09,9E+09]];
    CONST jointtarget jB_v13_t144 := [[45.0009,13.5374,47.9885,45.0009,46.166,-179.999],[9E+09,9E+09,9E+09,9E+09,9E+09,9E+09]];
    CONST jointtarget jBseed_v13_t144 := [[45.0009,13.5374,47.9885,45.0009,46.166,-179.999],[9E+09,9E+09,9E+09,9E+09,9E+09,9E+09]];

    CONST robtarget rA_v13_t145 := [[983.46,1103.96,351.653],[0.159979,-0.959864,-0.0681744,0.220047],[0,0,-2,0],[9E+09,9E+09,9E+09,9E+09,9E+09,9E+09]];
    CONST robtarget rB_v13_t145 := [[1514.11,1538.64,2797.39],[0.0241689,-0.261688,-0.327024,-0.907739],[0,1,-5,0],[9E+09,9E+09,9E+09,9E+09,9E+09,9E+09]];
    CONST robtarget rB_v13_t145_c4 := [[1514.11,1538.64,2797.39],[0.0241689,-0.261688,-0.327024,-0.907739],[0,-4,0,0],[9E+09,9E+09,9E+09,9E+09,9E+09,9E+09]];
    CONST robtarget rB_v13_t145_c5 := [[1514.11,1538.64,2797.39],[0.0241689,-0.261688,-0.327024,-0.907739],[0,0,0,0],[9E+09,9E+09,9E+09,9E+09,9E+09,9E+09]];
    CONST jointtarget jA_v13_t145 := [[45.0009,13.5374,47.9885,45.0009,46.166,-179.999],[9E+09,9E+09,9E+09,9E+09,9E+09,9E+09]];
    CONST jointtarget jB_v13_t145 := [[44.9995,29.7134,-64.4557,134.999,8.4579,-360.001],[9E+09,9E+09,9E+09,9E+09,9E+09,9E+09]];
    CONST jointtarget jBseed_v13_t145 := [[44.9995,29.7134,-64.4557,134.999,8.4579,-360.001],[9E+09,9E+09,9E+09,9E+09,9E+09,9E+09]];

    CONST robtarget rA_v13_t147 := [[2007.74,0.0318253,715.652],[0.597072,-0.292024,0.705031,-0.247303],[0,2,-3,0],[9E+09,9E+09,9E+09,9E+09,9E+09,9E+09]];
    CONST robtarget rB_v13_t147 := [[31.6778,2424.98,263.874],[0.0810362,-0.37401,-0.817272,-0.430832],[1,-2,-1,0],[9E+09,9E+09,9E+09,9E+09,9E+09,9E+09]];
    CONST robtarget rB_v13_t147_c6 := [[31.6778,2424.98,263.874],[0.0810362,-0.37401,-0.817272,-0.430832],[0,4,0,0],[9E+09,9E+09,9E+09,9E+09,9E+09,9E+09]];
    CONST jointtarget jA_v13_t147 := [[0.000956979,16.8297,30.3375,180.001,37.6879,-224.999],[9E+09,9E+09,9E+09,9E+09,9E+09,9E+09]];
    CONST jointtarget jB_v13_t147 := [[90.0005,47.7425,2.23639,-134.999,15.5718,-89.9995],[9E+09,9E+09,9E+09,9E+09,9E+09,9E+09]];
    CONST jointtarget jBseed_v13_t147 := [[90.0005,47.7425,2.2364,-134.999,15.5718,-89.9995],[9E+09,9E+09,9E+09,9E+09,9E+09,9E+09]];

    CONST robtarget rA_v13_t148 := [[31.6778,2424.98,263.874],[0.0810362,-0.37401,-0.817272,-0.430832],[1,-2,-1,0],[9E+09,9E+09,9E+09,9E+09,9E+09,9E+09]];
    CONST robtarget rB_v13_t148 := [[-0.000687608,-168.549,3019.24],[0.998319,-0.057957,3.42679E-6,-1.5789E-5],[-2,-3,2,0],[9E+09,9E+09,9E+09,9E+09,9E+09,9E+09]];
    CONST robtarget rB_v13_t148_c7 := [[-0.000687608,-168.549,3019.24],[0.998319,-0.057957,3.42679E-6,-1.5789E-5],[0,-4,4,0],[9E+09,9E+09,9E+09,9E+09,9E+09,9E+09]];
    CONST jointtarget jA_v13_t148 := [[90.0005,47.7425,2.23639,-134.999,15.5718,-89.9995],[9E+09,9E+09,9E+09,9E+09,9E+09,9E+09]];
    CONST jointtarget jB_v13_t148 := [[-90.0006,-46.1055,-10.8997,-180.001,39.6399,269.999],[9E+09,9E+09,9E+09,9E+09,9E+09,9E+09]];
    CONST jointtarget jBseed_v13_t148 := [[-90.0006,-46.1055,-10.8997,-180.001,39.6399,269.999],[9E+09,9E+09,9E+09,9E+09,9E+09,9E+09]];

    CONST robtarget rA_v13_t150 := [[0.00835412,392.696,3106.15],[0.529688,-0.46842,-0.468417,-0.529715],[0,-1,1,0],[9E+09,9E+09,9E+09,9E+09,9E+09,9E+09]];
    CONST robtarget rB_v13_t150 := [[1767.3,1767.24,55.4626],[0.441744,-0.336112,0.811427,0.182968],[0,1,1,0],[9E+09,9E+09,9E+09,9E+09,9E+09,9E+09]];
    CONST robtarget rB_v13_t150_c2 := [[1767.3,1767.24,55.4626],[0.441744,-0.336112,0.811427,0.182968],[0,0,-4,0],[9E+09,9E+09,9E+09,9E+09,9E+09,9E+09]];
    CONST robtarget rB_v13_t150_c5 := [[1767.3,1767.24,55.4626],[0.441744,-0.336112,0.811427,0.182968],[0,0,0,0],[9E+09,9E+09,9E+09,9E+09,9E+09,9E+09]];
    CONST jointtarget jA_v13_t150 := [[89.9991,-32.7458,-30.705,-0.000901862,56.4238,179.999],[9E+09,9E+09,9E+09,9E+09,9E+09,9E+09]];
    CONST jointtarget jB_v13_t150 := [[44.9992,58.0041,-4.9089,179.999,20.2228,179.999],[9E+09,9E+09,9E+09,9E+09,9E+09,9E+09]];
    CONST jointtarget jBseed_v13_t150 := [[44.9992,58.0041,-4.9089,179.999,20.2228,179.999],[9E+09,9E+09,9E+09,9E+09,9E+09,9E+09]];

    CONST robtarget rA_v13_t153 := [[-0.0456621,2850.01,1003.84],[0.254171,-0.65984,0.659847,0.254187],[1,0,-4,0],[9E+09,9E+09,9E+09,9E+09,9E+09,9E+09]];
    CONST robtarget rB_v13_t153 := [[-47.6013,1963.81,2611.81],[0.788239,-0.449679,0.0565546,0.416257],[0,1,-3,0],[9E+09,9E+09,9E+09,9E+09,9E+09,9E+09]];
    CONST robtarget rB_v13_t153_c2 := [[-47.6013,1963.81,2611.81],[0.788239,-0.449679,0.0565546,0.416257],[0,0,-4,0],[9E+09,9E+09,9E+09,9E+09,9E+09,9E+09]];
    CONST jointtarget jA_v13_t153 := [[90.0009,51.4707,-35.2595,0.000892354,31.6544,-359.999],[9E+09,9E+09,9E+09,9E+09,9E+09,9E+09]];
    CONST jointtarget jB_v13_t153 := [[89.9991,7.16147,-27.781,134.999,23.788,-180.001],[9E+09,9E+09,9E+09,9E+09,9E+09,9E+09]];
    CONST jointtarget jBseed_v13_t153 := [[89.9991,7.16148,-27.781,134.999,23.788,-180.001],[9E+09,9E+09,9E+09,9E+09,9E+09,9E+09]];

    CONST robtarget rA_v13_t154 := [[-47.6013,1963.81,2611.81],[0.788239,-0.449679,0.0565546,0.416257],[0,1,-3,0],[9E+09,9E+09,9E+09,9E+09,9E+09,9E+09]];
    CONST robtarget rB_v13_t154 := [[-851.318,851.307,3016.05],[0.691102,-0.211514,2.16484E-6,0.691115],[1,2,1,0],[9E+09,9E+09,9E+09,9E+09,9E+09,9E+09]];
    CONST robtarget rB_v13_t154_c1 := [[-851.318,851.307,3016.05],[0.691102,-0.211514,2.16484E-6,0.691115],[0,-4,-4,0],[9E+09,9E+09,9E+09,9E+09,9E+09,9E+09]];
    CONST jointtarget jA_v13_t154 := [[89.9991,7.16147,-27.781,134.999,23.788,-180.001],[9E+09,9E+09,9E+09,9E+09,9E+09,9E+09]];
    CONST jointtarget jB_v13_t154 := [[135,-14.5701,-23.4129,180,27.5948,135],[9E+09,9E+09,9E+09,9E+09,9E+09,9E+09]];
    CONST jointtarget jBseed_v13_t154 := [[135,-14.5701,-23.4129,180,27.5948,135],[9E+09,9E+09,9E+09,9E+09,9E+09,9E+09]];

    CONST robtarget rA_v13_t159 := [[1729.45,-1572.33,1894.97],[0.0141684,0.713328,-0.0265901,0.700183],[-1,1,1,0],[9E+09,9E+09,9E+09,9E+09,9E+09,9E+09]];
    CONST robtarget rB_v13_t159 := [[1526.55,-1553.12,620.862],[0.339535,0.679554,0.648254,-0.0518569],[-1,-1,0,0],[9E+09,9E+09,9E+09,9E+09,9E+09,9E+09]];
    CONST robtarget rB_v13_t159_c5 := [[1526.55,-1553.12,620.862],[0.339535,0.679554,0.648254,-0.0518569],[0,0,0,0],[9E+09,9E+09,9E+09,9E+09,9E+09,9E+09]];
    CONST jointtarget jA_v13_t159 := [[-44.9995,17.5622,-16.097,90.0005,41.6962,90.0005],[9E+09,9E+09,9E+09,9E+09,9E+09,9E+09]];
    CONST jointtarget jB_v13_t159 := [[-45.0005,26.2636,17.499,-45.0005,9.1464,89.9995],[9E+09,9E+09,9E+09,9E+09,9E+09,9E+09]];
    CONST jointtarget jBseed_v13_t159 := [[-45.0005,26.2636,17.499,-45.0005,9.1464,89.9995],[9E+09,9E+09,9E+09,9E+09,9E+09,9E+09]];

    CONST robtarget rA_v13_t167 := [[-537.007,579.743,3331.97],[0.023493,-0.180626,0.305344,0.934659],[1,-1,1,0],[9E+09,9E+09,9E+09,9E+09,9E+09,9E+09]];
    CONST robtarget rB_v13_t167 := [[35.551,173.515,2885.4],[0.668676,-0.203194,-0.0574588,-0.712939],[1,-2,-1,0],[9E+09,9E+09,9E+09,9E+09,9E+09,9E+09]];
    CONST robtarget rB_v13_t167_c5 := [[35.551,173.515,2885.4],[0.668676,-0.203194,-0.0574588,-0.712939],[0,0,0,0],[9E+09,9E+09,9E+09,9E+09,9E+09,9E+09]];
    CONST robtarget rB_v13_t167_c8 := [[35.551,173.515,2885.4],[0.668676,-0.203194,-0.0574588,-0.712939],[0,0,4,0],[9E+09,9E+09,9E+09,9E+09,9E+09,9E+09]];
    CONST jointtarget jA_v13_t167 := [[135.001,-12.0505,-48.0941,-44.9993,14.832,90.0007],[9E+09,9E+09,9E+09,9E+09,9E+09,9E+09]];
    CONST jointtarget jB_v13_t167 := [[90.0006,-53.5032,-2.69113,-134.999,17.5219,-44.9994],[9E+09,9E+09,9E+09,9E+09,9E+09,9E+09]];
    CONST jointtarget jBseed_v13_t167 := [[90.0006,-53.5032,-2.69112,-134.999,17.5219,-44.9994],[9E+09,9E+09,9E+09,9E+09,9E+09,9E+09]];

    CONST robtarget rA_v13_t168 := [[35.551,173.515,2885.4],[0.668676,-0.203194,-0.0574588,-0.712939],[1,-2,-1,0],[9E+09,9E+09,9E+09,9E+09,9E+09,9E+09]];
    CONST robtarget rB_v13_t168 := [[793.493,-595.149,3244.1],[0.452793,-0.522036,0.068001,-0.719606],[-1,-4,1,0],[9E+09,9E+09,9E+09,9E+09,9E+09,9E+09]];
    CONST robtarget rB_v13_t168_c4 := [[793.493,-595.149,3244.1],[0.452793,-0.522036,0.068001,-0.719606],[0,-4,0,0],[9E+09,9E+09,9E+09,9E+09,9E+09,9E+09]];
    CONST robtarget rB_v13_t168_c5 := [[793.493,-595.149,3244.1],[0.452793,-0.522036,0.068001,-0.719606],[0,0,0,0],[9E+09,9E+09,9E+09,9E+09,9E+09,9E+09]];
    CONST jointtarget jA_v13_t168 := [[90.0006,-53.5032,-2.69113,-134.999,17.5219,-44.9994],[9E+09,9E+09,9E+09,9E+09,9E+09,9E+09]];
    CONST jointtarget jB_v13_t168 := [[-45.0007,-5.56475,-49.6414,-270.001,57.1288,179.999],[9E+09,9E+09,9E+09,9E+09,9E+09,9E+09]];
    CONST jointtarget jBseed_v13_t168 := [[-45.0007,-5.56474,-49.6414,-270.001,57.1288,179.999],[9E+09,9E+09,9E+09,9E+09,9E+09,9E+09]];

    CONST robtarget rA_v13_t171 := [[-375.162,-375.157,3315.91],[0.998794,0.0347135,-0.0347109,-1.13746E-5],[-2,1,3,0],[9E+09,9E+09,9E+09,9E+09,9E+09,9E+09]];
    CONST robtarget rB_v13_t171 := [[60.3441,-2778.86,702.129],[0.0920256,0.371449,-0.657421,0.649119],[-1,-3,1,0],[9E+09,9E+09,9E+09,9E+09,9E+09,9E+09]];
    CONST robtarget rB_v13_t171_c5 := [[60.3441,-2778.86,702.129],[0.0920256,0.371449,-0.657421,0.649119],[0,0,0,0],[9E+09,9E+09,9E+09,9E+09,9E+09,9E+09]];
    CONST jointtarget jA_v13_t171 := [[-135,-21.554,-38.243,180,24.5753,315],[9E+09,9E+09,9E+09,9E+09,9E+09,9E+09]];
    CONST jointtarget jB_v13_t171 := [[-89.9996,51.8186,-20.3699,-225,30.7205,90.0004],[9E+09,9E+09,9E+09,9E+09,9E+09,9E+09]];
    CONST jointtarget jBseed_v13_t171 := [[-89.9996,51.8186,-20.3699,-225,30.7205,90.0004],[9E+09,9E+09,9E+09,9E+09,9E+09,9E+09]];

    CONST robtarget rA_v13_t174 := [[33.1237,2104.46,2700.8],[0.0527459,0.0852185,0.435832,0.894431],[1,-2,2,0],[9E+09,9E+09,9E+09,9E+09,9E+09,9E+09]];
    CONST robtarget rB_v13_t174 := [[-1227.25,1159.65,3106.61],[0.63746,-0.245423,-0.13471,0.71782],[1,-3,2,0],[9E+09,9E+09,9E+09,9E+09,9E+09,9E+09]];
    CONST robtarget rB_v13_t174_c4 := [[-1227.25,1159.65,3106.61],[0.63746,-0.245423,-0.13471,0.71782],[0,-4,0,0],[9E+09,9E+09,9E+09,9E+09,9E+09,9E+09]];
    CONST robtarget rB_v13_t174_c5 := [[-1227.25,1159.65,3106.61],[0.63746,-0.245423,-0.13471,0.71782],[0,0,0,0],[9E+09,9E+09,9E+09,9E+09,9E+09,9E+09]];
    CONST jointtarget jA_v13_t174 := [[90.0004,18.7378,-45.2178,-135,16.2969,225],[9E+09,9E+09,9E+09,9E+09,9E+09,9E+09]];
    CONST jointtarget jB_v13_t174 := [[135.001,16.7821,-61.0556,-224.999,23.8649,180.001],[9E+09,9E+09,9E+09,9E+09,9E+09,9E+09]];
    CONST jointtarget jBseed_v13_t174 := [[135.001,16.7821,-61.0556,-224.999,23.8649,180.001],[9E+09,9E+09,9E+09,9E+09,9E+09,9E+09]];

    CONST robtarget rA_v13_t176 := [[181.94,-268.656,3362.57],[0.0382584,-0.127432,-0.136712,0.981635],[-1,-2,4,0],[9E+09,9E+09,9E+09,9E+09,9E+09,9E+09]];
    CONST robtarget rB_v13_t176 := [[1926.8,1926.78,1896.74],[0.648407,-0.398906,-2.45054E-6,-0.648416],[0,1,-4,0],[9E+09,9E+09,9E+09,9E+09,9E+09,9E+09]];
    CONST robtarget rB_v13_t176_c4 := [[1926.8,1926.78,1896.74],[0.648407,-0.398906,-2.45054E-6,-0.648416],[0,-4,0,0],[9E+09,9E+09,9E+09,9E+09,9E+09,9E+09]];
    CONST jointtarget jA_v13_t176 := [[-44.9992,-22.356,-44.4798,-134.999,31.2845,360.001],[9E+09,9E+09,9E+09,9E+09,9E+09,9E+09]];
    CONST jointtarget jB_v13_t176 := [[44.9997,41.8647,-44.7932,180,40.0519,-315],[9E+09,9E+09,9E+09,9E+09,9E+09,9E+09]];
    CONST jointtarget jBseed_v13_t176 := [[44.9997,41.8647,-44.7932,180,40.0519,-315],[9E+09,9E+09,9E+09,9E+09,9E+09,9E+09]];

    CONST robtarget rA_v13_t177 := [[1926.8,1926.78,1896.74],[0.648407,-0.398906,-2.45054E-6,-0.648416],[0,1,-4,0],[9E+09,9E+09,9E+09,9E+09,9E+09,9E+09]];
    CONST robtarget rB_v13_t177 := [[0.0188833,-1684.03,2981.44],[0.382096,0.0209191,-0.0505156,0.922504],[-1,2,0,0],[9E+09,9E+09,9E+09,9E+09,9E+09,9E+09]];
    CONST robtarget rB_v13_t177_c2 := [[0.0188833,-1684.03,2981.44],[0.382096,0.0209191,-0.0505156,0.922504],[0,0,-4,0],[9E+09,9E+09,9E+09,9E+09,9E+09,9E+09]];
    CONST robtarget rB_v13_t177_c5 := [[0.0188833,-1684.03,2981.44],[0.382096,0.0209191,-0.0505156,0.922504],[0,0,0,0],[9E+09,9E+09,9E+09,9E+09,9E+09,9E+09]];
    CONST jointtarget jA_v13_t177 := [[44.9997,41.8647,-44.7932,180,40.0519,-315],[9E+09,9E+09,9E+09,9E+09,9E+09,9E+09]];
    CONST jointtarget jB_v13_t177 := [[-89.9993,9.40275,-43.8609,180.001,49.2734,45.0007],[9E+09,9E+09,9E+09,9E+09,9E+09,9E+09]];
    CONST jointtarget jBseed_v13_t177 := [[-89.9993,9.40276,-43.8609,180.001,49.2734,45.0007],[9E+09,9E+09,9E+09,9E+09,9E+09,9E+09]];

    CONST robtarget rA_v13_t178 := [[0.0188833,-1684.03,2981.44],[0.382096,0.0209191,-0.0505156,0.922504],[-1,2,0,0],[9E+09,9E+09,9E+09,9E+09,9E+09,9E+09]];
    CONST robtarget rB_v13_t178 := [[-51.6131,2106.49,2267.54],[0.736335,-0.542266,-0.354113,-0.195862],[0,-4,1,0],[9E+09,9E+09,9E+09,9E+09,9E+09,9E+09]];
    CONST robtarget rB_v13_t178_c2 := [[-51.6131,2106.49,2267.54],[0.736335,-0.542266,-0.354113,-0.195862],[0,0,-4,0],[9E+09,9E+09,9E+09,9E+09,9E+09,9E+09]];
    CONST jointtarget jA_v13_t178 := [[-89.9993,9.40275,-43.8609,180.001,49.2734,45.0007],[9E+09,9E+09,9E+09,9E+09,9E+09,9E+09]];
    CONST jointtarget jB_v13_t178 := [[89.9999,7.11386,-16.8667,-270,18.0035,135],[9E+09,9E+09,9E+09,9E+09,9E+09,9E+09]];
    CONST jointtarget jBseed_v13_t178 := [[89.9999,7.11386,-16.8667,-270,18.0035,135],[9E+09,9E+09,9E+09,9E+09,9E+09,9E+09]];

    CONST robtarget rA_v13_t179 := [[-51.6131,2106.49,2267.54],[0.736335,-0.542266,-0.354113,-0.195862],[0,-4,1,0],[9E+09,9E+09,9E+09,9E+09,9E+09,9E+09]];
    CONST robtarget rB_v13_t179 := [[1445.43,1334.37,824.632],[0.40796,-0.550386,0.694482,-0.21986],[0,-2,0,0],[9E+09,9E+09,9E+09,9E+09,9E+09,9E+09]];
    CONST robtarget rB_v13_t179_c5 := [[1445.43,1334.37,824.632],[0.40796,-0.550386,0.694482,-0.21986],[0,0,0,0],[9E+09,9E+09,9E+09,9E+09,9E+09,9E+09]];
    CONST jointtarget jA_v13_t179 := [[89.9999,7.11386,-16.8667,-270,18.0035,135],[9E+09,9E+09,9E+09,9E+09,9E+09,9E+09]];
    CONST jointtarget jB_v13_t179 := [[44.9996,11.4902,28.7783,-90.0004,28.0471,44.9996],[9E+09,9E+09,9E+09,9E+09,9E+09,9E+09]];
    CONST jointtarget jBseed_v13_t179 := [[44.9996,11.4902,28.7783,-90.0004,28.0471,44.9996],[9E+09,9E+09,9E+09,9E+09,9E+09,9E+09]];

    CONST robtarget rA_v13_t180 := [[1445.43,1334.37,824.632],[0.40796,-0.550386,0.694482,-0.21986],[0,-2,0,0],[9E+09,9E+09,9E+09,9E+09,9E+09,9E+09]];
    CONST robtarget rB_v13_t180 := [[1456.15,-1373.77,2949.02],[0.302727,0.258096,0.0730139,0.914555],[-1,-3,0,0],[9E+09,9E+09,9E+09,9E+09,9E+09,9E+09]];
    CONST robtarget rB_v13_t180_c4 := [[1456.15,-1373.77,2949.02],[0.302727,0.258096,0.0730139,0.914555],[0,-4,0,0],[9E+09,9E+09,9E+09,9E+09,9E+09,9E+09]];
    CONST robtarget rB_v13_t180_c5 := [[1456.15,-1373.77,2949.02],[0.302727,0.258096,0.0730139,0.914555],[0,0,0,0],[9E+09,9E+09,9E+09,9E+09,9E+09,9E+09]];
    CONST jointtarget jA_v13_t180 := [[44.9996,11.4902,28.7783,-90.0004,28.0471,44.9996],[9E+09,9E+09,9E+09,9E+09,9E+09,9E+09]];
    CONST jointtarget jB_v13_t180 := [[-45.0009,35.2287,-79.3652,-225.001,29.5761,44.9991],[9E+09,9E+09,9E+09,9E+09,9E+09,9E+09]];
    CONST jointtarget jBseed_v13_t180 := [[-45.0009,35.2287,-79.3652,-225.001,29.5761,44.9991],[9E+09,9E+09,9E+09,9E+09,9E+09,9E+09]];

    CONST robtarget rA_v13_t182 := [[-1657.55,1580.58,884.848],[0.348295,-0.283518,-0.893351,0.0152197],[1,0,1,0],[9E+09,9E+09,9E+09,9E+09,9E+09,9E+09]];
    CONST robtarget rB_v13_t182 := [[-38.062,1657.56,1581.01],[0.615029,-0.682635,-0.361358,-0.158648],[1,-3,-3,0],[9E+09,9E+09,9E+09,9E+09,9E+09,9E+09]];
    CONST robtarget rB_v13_t182_c4 := [[-38.062,1657.56,1581.01],[0.615029,-0.682635,-0.361358,-0.158648],[0,-4,0,0],[9E+09,9E+09,9E+09,9E+09,9E+09,9E+09]];
    CONST robtarget rB_v13_t182_c5 := [[-38.062,1657.56,1581.01],[0.615029,-0.682635,-0.361358,-0.158648],[0,0,0,0],[9E+09,9E+09,9E+09,9E+09,9E+09,9E+09]];
    CONST jointtarget jA_v13_t182 := [[135.001,24.7401,8.29463,45.0009,27.4264,135.001],[9E+09,9E+09,9E+09,9E+09,9E+09,9E+09]];
    CONST jointtarget jB_v13_t182 := [[90.0001,-19.7375,31.1786,-270,13.173,-225],[9E+09,9E+09,9E+09,9E+09,9E+09,9E+09]];
    CONST jointtarget jBseed_v13_t182 := [[90.0001,-19.7375,31.1786,-270,13.173,-225],[9E+09,9E+09,9E+09,9E+09,9E+09,9E+09]];

    CONST robtarget rA_v13_t183 := [[-38.062,1657.56,1581.01],[0.615029,-0.682635,-0.361358,-0.158648],[1,-3,-3,0],[9E+09,9E+09,9E+09,9E+09,9E+09,9E+09]];
    CONST robtarget rB_v13_t183 := [[699.984,633.226,3136.18],[0.0492623,0.428135,0.236196,0.87091],[0,-1,-2,0],[9E+09,9E+09,9E+09,9E+09,9E+09,9E+09]];
    CONST robtarget rB_v13_t183_c2 := [[699.984,633.226,3136.18],[0.0492623,0.428135,0.236196,0.87091],[0,0,-4,0],[9E+09,9E+09,9E+09,9E+09,9E+09,9E+09]];
    CONST jointtarget jA_v13_t183 := [[90.0001,-19.7375,31.1786,-270,13.173,-225],[9E+09,9E+09,9E+09,9E+09,9E+09,9E+09]];
    CONST jointtarget jB_v13_t183 := [[45.0002,-18.2617,-31.8357,-44.9998,23.5646,-180],[9E+09,9E+09,9E+09,9E+09,9E+09,9E+09]];
    CONST jointtarget jBseed_v13_t183 := [[45.0002,-18.2617,-31.8357,-44.9998,23.5646,-180],[9E+09,9E+09,9E+09,9E+09,9E+09,9E+09]];

    CONST robtarget rA_v13_t184 := [[699.984,633.226,3136.18],[0.0492623,0.428135,0.236196,0.87091],[0,-1,-2,0],[9E+09,9E+09,9E+09,9E+09,9E+09,9E+09]];
    CONST robtarget rB_v13_t184 := [[-61.6846,538.639,3476.67],[0.887603,-0.201759,-0.117825,0.396953],[1,1,-2,0],[9E+09,9E+09,9E+09,9E+09,9E+09,9E+09]];
    CONST robtarget rB_v13_t184_c4 := [[-61.6846,538.639,3476.67],[0.887603,-0.201759,-0.117825,0.396953],[0,-4,0,0],[9E+09,9E+09,9E+09,9E+09,9E+09,9E+09]];
    CONST robtarget rB_v13_t184_c5 := [[-61.6846,538.639,3476.67],[0.887603,-0.201759,-0.117825,0.396953],[0,0,0,0],[9E+09,9E+09,9E+09,9E+09,9E+09,9E+09]];
    CONST jointtarget jA_v13_t184 := [[45.0002,-18.2617,-31.8357,-44.9998,23.5646,-180],[9E+09,9E+09,9E+09,9E+09,9E+09,9E+09]];
    CONST jointtarget jB_v13_t184 := [[90.0005,-3.81414,-69.6412,90.0004,21.6749,-134.999],[9E+09,9E+09,9E+09,9E+09,9E+09,9E+09]];
    CONST jointtarget jBseed_v13_t184 := [[90.0005,-3.81421,-69.6411,90.0005,21.6749,-134.999],[9E+09,9E+09,9E+09,9E+09,9E+09,9E+09]];

    CONST robtarget rA_v13_t187 := [[-30.46,2921.9,902.083],[0.498636,-0.773938,0.263702,0.287825],[0,-4,-2,0],[9E+09,9E+09,9E+09,9E+09,9E+09,9E+09]];
    CONST robtarget rB_v13_t187 := [[2151.62,40.8526,711.969],[0.298293,-0.808416,0.281584,-0.422133],[0,-3,1,0],[9E+09,9E+09,9E+09,9E+09,9E+09,9E+09]];
    CONST robtarget rB_v13_t187_c1 := [[2151.62,40.8526,711.969],[0.298293,-0.808416,0.281584,-0.422133],[0,-4,-4,0],[9E+09,9E+09,9E+09,9E+09,9E+09,9E+09]];
    CONST jointtarget jA_v13_t187 := [[89.9995,55.7115,-35.6642,-270,10.5179,-135],[9E+09,9E+09,9E+09,9E+09,9E+09,9E+09]];
    CONST jointtarget jB_v13_t187 := [[0.000328933,22.3743,20.9348,-225,20.2338,90.0003],[9E+09,9E+09,9E+09,9E+09,9E+09,9E+09]];
    CONST jointtarget jBseed_v13_t187 := [[0.000328959,22.3743,20.9348,-225,20.2338,90.0003],[9E+09,9E+09,9E+09,9E+09,9E+09,9E+09]];

    CONST robtarget rA_v13_t188 := [[2151.62,40.8526,711.969],[0.298293,-0.808416,0.281584,-0.422133],[0,-3,1,0],[9E+09,9E+09,9E+09,9E+09,9E+09,9E+09]];
    CONST robtarget rB_v13_t188 := [[2595.98,54.1421,1846.79],[0.798602,-0.116648,0.578265,0.119323],[-1,1,2,0],[9E+09,9E+09,9E+09,9E+09,9E+09,9E+09]];
    CONST robtarget rB_v13_t188_c1 := [[2595.98,54.1421,1846.79],[0.798602,-0.116648,0.578265,0.119323],[0,-4,-4,0],[9E+09,9E+09,9E+09,9E+09,9E+09,9E+09]];
    CONST robtarget rB_v13_t188_c4 := [[2595.98,54.1421,1846.79],[0.798602,-0.116648,0.578265,0.119323],[0,-4,0,0],[9E+09,9E+09,9E+09,9E+09,9E+09,9E+09]];
    CONST jointtarget jA_v13_t188 := [[0.000328933,22.3743,20.9348,-225,20.2338,90.0003],[9E+09,9E+09,9E+09,9E+09,9E+09,9E+09]];
    CONST jointtarget jB_v13_t188 := [[-0.000414314,30.8744,-29.5703,135,27.3,225],[9E+09,9E+09,9E+09,9E+09,9E+09,9E+09]];
    CONST jointtarget jBseed_v13_t188 := [[-0.000414289,30.8744,-29.5703,135,27.3,225],[9E+09,9E+09,9E+09,9E+09,9E+09,9E+09]];

    CONST robtarget rA_v13_t189 := [[2595.98,54.1421,1846.79],[0.798602,-0.116648,0.578265,0.119323],[-1,1,2,0],[9E+09,9E+09,9E+09,9E+09,9E+09,9E+09]];
    CONST robtarget rB_v13_t189 := [[-13.4206,-2934.15,740.094],[0.520367,0.761897,0.291958,-0.251977],[-2,2,-3,0],[9E+09,9E+09,9E+09,9E+09,9E+09,9E+09]];
    CONST robtarget rB_v13_t189_c4 := [[-13.4206,-2934.15,740.094],[0.520367,0.761897,0.291958,-0.251977],[0,-4,0,0],[9E+09,9E+09,9E+09,9E+09,9E+09,9E+09]];
    CONST robtarget rB_v13_t189_c5 := [[-13.4206,-2934.15,740.094],[0.520367,0.761897,0.291958,-0.251977],[0,0,0,0],[9E+09,9E+09,9E+09,9E+09,9E+09,9E+09]];
    CONST jointtarget jA_v13_t189 := [[-0.000414314,30.8744,-29.5703,135,27.3,225],[9E+09,9E+09,9E+09,9E+09,9E+09,9E+09]];
    CONST jointtarget jB_v13_t189 := [[-90.0009,59.2309,-35.2001,224.999,6.5041,-180.001],[9E+09,9E+09,9E+09,9E+09,9E+09,9E+09]];
    CONST jointtarget jBseed_v13_t189 := [[-90.0009,59.2309,-35.2,224.999,6.5041,-180.001],[9E+09,9E+09,9E+09,9E+09,9E+09,9E+09]];

    CONST robtarget rA_v13_t190 := [[-13.4206,-2934.15,740.094],[0.520367,0.761897,0.291958,-0.251977],[-2,2,-3,0],[9E+09,9E+09,9E+09,9E+09,9E+09,9E+09]];
    CONST robtarget rB_v13_t190 := [[-199.244,-199.249,3190.85],[0.373465,-0.0834226,-0.201396,0.901667],[-2,-2,1,0],[9E+09,9E+09,9E+09,9E+09,9E+09,9E+09]];
    CONST robtarget rB_v13_t190_c2 := [[-199.244,-199.249,3190.85],[0.373465,-0.0834226,-0.201396,0.901667],[0,0,-4,0],[9E+09,9E+09,9E+09,9E+09,9E+09,9E+09]];
    CONST robtarget rB_v13_t190_c5 := [[-199.244,-199.249,3190.85],[0.373465,-0.0834226,-0.201396,0.901667],[0,0,0,0],[9E+09,9E+09,9E+09,9E+09,9E+09,9E+09]];
    CONST jointtarget jA_v13_t190 := [[-90.0009,59.2309,-35.2001,224.999,6.5041,-180.001],[9E+09,9E+09,9E+09,9E+09,9E+09,9E+09]];
    CONST jointtarget jB_v13_t190 := [[-134.999,-35.8257,-26.317,-179.999,2.67526,90.0006],[9E+09,9E+09,9E+09,9E+09,9E+09,9E+09]];
    CONST jointtarget jBseed_v13_t190 := [[-134.999,-35.8257,-26.317,-179.999,2.67525,90.0006],[9E+09,9E+09,9E+09,9E+09,9E+09,9E+09]];

    CONST robtarget rA_v13_t193 := [[-697.848,-697.862,2965.67],[0.922837,0.0440026,-0.0182315,-0.382234],[-2,2,3,0],[9E+09,9E+09,9E+09,9E+09,9E+09,9E+09]];
    CONST robtarget rB_v13_t193 := [[2331.06,0.0127871,387.445],[0.0367367,-0.919612,0.380918,-0.0886846],[0,0,2,0],[9E+09,9E+09,9E+09,9E+09,9E+09,9E+09]];
    CONST robtarget rB_v13_t193_c8 := [[2331.06,0.0127871,387.445],[0.0367367,-0.919612,0.380918,-0.0886846],[0,0,4,0],[9E+09,9E+09,9E+09,9E+09,9E+09,9E+09]];
    CONST jointtarget jA_v13_t193 := [[-134.999,-23.7623,-13.9268,180.001,46.8508,270.001],[9E+09,9E+09,9E+09,9E+09,9E+09,9E+09]];
    CONST jointtarget jB_v13_t193 := [[0.000302251,41.6999,3.39487,0.000301556,33.8884,225],[9E+09,9E+09,9E+09,9E+09,9E+09,9E+09]];
    CONST jointtarget jBseed_v13_t193 := [[0.000302225,41.6999,3.39487,0.000302225,33.8884,225],[9E+09,9E+09,9E+09,9E+09,9E+09,9E+09]];

    CONST robtarget rA_v13_t194 := [[2331.06,0.0127871,387.445],[0.0367367,-0.919612,0.380918,-0.0886846],[0,0,2,0],[9E+09,9E+09,9E+09,9E+09,9E+09,9E+09]];
    CONST robtarget rB_v13_t194 := [[1205.57,1032.95,-168.256],[0.070505,-0.624956,0.668282,-0.397313],[0,3,0,0],[9E+09,9E+09,9E+09,9E+09,9E+09,9E+09]];
    CONST robtarget rB_v13_t194_c5 := [[1205.57,1032.95,-168.256],[0.070505,-0.624956,0.668282,-0.397313],[0,0,0,0],[9E+09,9E+09,9E+09,9E+09,9E+09,9E+09]];
    CONST jointtarget jA_v13_t194 := [[0.000302251,41.6999,3.39487,0.000301556,33.8884,225],[9E+09,9E+09,9E+09,9E+09,9E+09,9E+09]];
    CONST jointtarget jB_v13_t194 := [[45.0005,46.3619,34.8207,270,46.968,45.0005],[9E+09,9E+09,9E+09,9E+09,9E+09,9E+09]];
    CONST jointtarget jBseed_v13_t194 := [[45.0005,46.3619,34.8207,270,46.968,45.0005],[9E+09,9E+09,9E+09,9E+09,9E+09,9E+09]];

    CONST robtarget rA_v13_t195 := [[1205.57,1032.95,-168.256],[0.070505,-0.624956,0.668282,-0.397313],[0,3,0,0],[9E+09,9E+09,9E+09,9E+09,9E+09,9E+09]];
    CONST robtarget rB_v13_t195 := [[-19.8759,1637.49,511.186],[0.220905,-0.669058,-0.695527,-0.140728],[1,0,-3,0],[9E+09,9E+09,9E+09,9E+09,9E+09,9E+09]];
    CONST robtarget rB_v13_t195_c5 := [[-19.8759,1637.49,511.186],[0.220905,-0.669058,-0.695527,-0.140728],[0,0,0,0],[9E+09,9E+09,9E+09,9E+09,9E+09,9E+09]];
    CONST jointtarget jA_v13_t195 := [[45.0005,46.3619,34.8207,270,46.968,45.0005],[9E+09,9E+09,9E+09,9E+09,9E+09,9E+09]];
    CONST jointtarget jB_v13_t195 := [[90.0002,7.86828,45.5883,45.0002,9.68657,-225],[9E+09,9E+09,9E+09,9E+09,9E+09,9E+09]];
    CONST jointtarget jBseed_v13_t195 := [[90.0002,7.86829,45.5882,45.0002,9.68657,-225],[9E+09,9E+09,9E+09,9E+09,9E+09,9E+09]];

    CONST robtarget rA_v13_t196 := [[-19.8759,1637.49,511.186],[0.220905,-0.669058,-0.695527,-0.140728],[1,0,-3,0],[9E+09,9E+09,9E+09,9E+09,9E+09,9E+09]];
    CONST robtarget rB_v13_t196 := [[1376.01,1363.72,2808.48],[0.348621,0.202538,0.430007,0.807797],[0,-2,2,0],[9E+09,9E+09,9E+09,9E+09,9E+09,9E+09]];
    CONST robtarget rB_v13_t196_c1 := [[1376.01,1363.72,2808.48],[0.348621,0.202538,0.430007,0.807797],[0,-4,-4,0],[9E+09,9E+09,9E+09,9E+09,9E+09,9E+09]];
    CONST robtarget rB_v13_t196_c2 := [[1376.01,1363.72,2808.48],[0.348621,0.202538,0.430007,0.807797],[0,0,-4,0],[9E+09,9E+09,9E+09,9E+09,9E+09,9E+09]];
    CONST jointtarget jA_v13_t196 := [[90.0002,7.86828,45.5883,45.0002,9.68657,-225],[9E+09,9E+09,9E+09,9E+09,9E+09,9E+09]];
    CONST jointtarget jB_v13_t196 := [[44.9997,12.5193,-42.8254,-135,4.21704,225],[9E+09,9E+09,9E+09,9E+09,9E+09,9E+09]];
    CONST jointtarget jBseed_v13_t196 := [[44.9997,12.5193,-42.8254,-135,4.21705,225],[9E+09,9E+09,9E+09,9E+09,9E+09,9E+09]];

    CONST robtarget rA_v13_t197 := [[1376.01,1363.72,2808.48],[0.348621,0.202538,0.430007,0.807797],[0,-2,2,0],[9E+09,9E+09,9E+09,9E+09,9E+09,9E+09]];
    CONST robtarget rB_v13_t197 := [[0.00233228,-235.495,3361.07],[0.702804,-0.0777345,0.0777287,0.702838],[-1,-2,-4,0],[9E+09,9E+09,9E+09,9E+09,9E+09,9E+09]];
    CONST robtarget rB_v13_t197_c7 := [[0.00233228,-235.495,3361.07],[0.702804,-0.0777345,0.0777287,0.702838],[0,-4,4,0],[9E+09,9E+09,9E+09,9E+09,9E+09,9E+09]];
    CONST robtarget rB_v13_t197_c8 := [[0.00233228,-235.495,3361.07],[0.702804,-0.0777345,0.0777287,0.702838],[0,0,4,0],[9E+09,9E+09,9E+09,9E+09,9E+09,9E+09]];
    CONST jointtarget jA_v13_t197 := [[44.9997,12.5193,-42.8254,-135,4.21704,225],[9E+09,9E+09,9E+09,9E+09,9E+09,9E+09]];
    CONST jointtarget jB_v13_t197 := [[-89.999,-24.0992,-43.3293,-179.999,35.1939,-359.999],[9E+09,9E+09,9E+09,9E+09,9E+09,9E+09]];
    CONST jointtarget jBseed_v13_t197 := [[-89.999,-24.0992,-43.3293,-179.999,35.1939,-359.999],[9E+09,9E+09,9E+09,9E+09,9E+09,9E+09]];

    CONST robtarget rA_v13_t200 := [[-572.033,572.019,2517.87],[0.320044,0.209825,-0.506569,-0.772615],[1,0,1,0],[9E+09,9E+09,9E+09,9E+09,9E+09,9E+09]];
    CONST robtarget rB_v13_t200 := [[32.706,158.336,3170.29],[0.855085,-0.234838,-0.17524,0.427752],[0,-3,2,0],[9E+09,9E+09,9E+09,9E+09,9E+09,9E+09]];
    CONST robtarget rB_v13_t200_c2 := [[32.706,158.336,3170.29],[0.855085,-0.234838,-0.17524,0.427752],[0,0,-4,0],[9E+09,9E+09,9E+09,9E+09,9E+09,9E+09]];
    CONST robtarget rB_v13_t200_c5 := [[32.706,158.336,3170.29],[0.855085,-0.234838,-0.17524,0.427752],[0,0,0,0],[9E+09,9E+09,9E+09,9E+09,9E+09,9E+09]];
    CONST jointtarget jA_v13_t200 := [[135.001,-48.0905,13.9918,0.000669506,10.6003,90.0006],[9E+09,9E+09,9E+09,9E+09,9E+09,9E+09]];
    CONST jointtarget jB_v13_t200 := [[44.9994,-37.243,-25.837,-225.001,48.7881,224.999],[9E+09,9E+09,9E+09,9E+09,9E+09,9E+09]];
    CONST jointtarget jBseed_v13_t200 := [[44.9994,-37.243,-25.837,-225.001,48.7881,224.999],[9E+09,9E+09,9E+09,9E+09,9E+09,9E+09]];

    CONST robtarget rA_v13_t201 := [[32.706,158.336,3170.29],[0.855085,-0.234838,-0.17524,0.427752],[0,-3,2,0],[9E+09,9E+09,9E+09,9E+09,9E+09,9E+09]];
    CONST robtarget rB_v13_t201 := [[943.945,94.6594,3183.68],[0.467504,-0.134818,-0.264664,-0.832596],[0,-3,-3,0],[9E+09,9E+09,9E+09,9E+09,9E+09,9E+09]];
    CONST robtarget rB_v13_t201_c4 := [[943.945,94.6594,3183.68],[0.467504,-0.134818,-0.264664,-0.832596],[0,-4,0,0],[9E+09,9E+09,9E+09,9E+09,9E+09,9E+09]];
    CONST jointtarget jA_v13_t201 := [[44.9994,-37.243,-25.837,-225.001,48.7881,224.999],[9E+09,9E+09,9E+09,9E+09,9E+09,9E+09]];
    CONST jointtarget jB_v13_t201 := [[0.000501121,-13.2224,-34.9065,-224.999,53.278,-270],[9E+09,9E+09,9E+09,9E+09,9E+09,9E+09]];
    CONST jointtarget jBseed_v13_t201 := [[0.000501144,-13.2225,-34.9065,-224.999,53.278,-270],[9E+09,9E+09,9E+09,9E+09,9E+09,9E+09]];

    CONST robtarget rA_v13_t202 := [[943.945,94.6594,3183.68],[0.467504,-0.134818,-0.264664,-0.832596],[0,-3,-3,0],[9E+09,9E+09,9E+09,9E+09,9E+09,9E+09]];
    CONST robtarget rB_v13_t202 := [[1435.84,1446.09,1888.33],[0.496028,-0.72753,-0.014835,-0.473747],[0,1,1,0],[9E+09,9E+09,9E+09,9E+09,9E+09,9E+09]];
    CONST robtarget rB_v13_t202_c1 := [[1435.84,1446.09,1888.33],[0.496028,-0.72753,-0.014835,-0.473747],[0,-4,-4,0],[9E+09,9E+09,9E+09,9E+09,9E+09,9E+09]];
    CONST jointtarget jA_v13_t202 := [[0.000501121,-13.2224,-34.9065,-224.999,53.278,-270],[9E+09,9E+09,9E+09,9E+09,9E+09,9E+09]];
    CONST jointtarget jB_v13_t202 := [[45.0006,-0.272835,3.66069,90.0007,2.47932,135.001],[9E+09,9E+09,9E+09,9E+09,9E+09,9E+09]];
    CONST jointtarget jBseed_v13_t202 := [[45.0006,-0.272835,3.66069,90.0006,2.47932,135.001],[9E+09,9E+09,9E+09,9E+09,9E+09,9E+09]];

    CONST robtarget rA_v13_t206 := [[-369.496,-446.533,2454.18],[0.899671,0.324737,0.0275528,-0.290481],[-2,-3,3,0],[9E+09,9E+09,9E+09,9E+09,9E+09,9E+09]];
    CONST robtarget rB_v13_t206 := [[385.549,-262.482,2605.12],[0.118021,-0.268428,-0.097868,-0.95102],[-1,-3,-4,0],[9E+09,9E+09,9E+09,9E+09,9E+09,9E+09]];
    CONST robtarget rB_v13_t206_c4 := [[385.549,-262.482,2605.12],[0.118021,-0.268428,-0.097868,-0.95102],[0,-4,0,0],[9E+09,9E+09,9E+09,9E+09,9E+09,9E+09]];
    CONST jointtarget jA_v13_t206 := [[-134.999,-59.0185,22.7796,-224.999,27.4667,315.001],[9E+09,9E+09,9E+09,9E+09,9E+09,9E+09]];
    CONST jointtarget jB_v13_t206 := [[-45.0006,-55.8214,14.821,-225.001,47.4734,-270.001],[9E+09,9E+09,9E+09,9E+09,9E+09,9E+09]];
    CONST jointtarget jBseed_v13_t206 := [[-45.0006,-55.8214,14.821,-225.001,47.4734,-270.001],[9E+09,9E+09,9E+09,9E+09,9E+09,9E+09]];

    CONST robtarget rA_v13_t208 := [[-868.473,-1062.76,2627.18],[0.0585679,0.18302,-0.585874,0.78729],[-2,0,-3,0],[9E+09,9E+09,9E+09,9E+09,9E+09,9E+09]];
    CONST robtarget rB_v13_t208 := [[173.996,-336.828,2929.77],[0.770747,0.436735,0.13255,-0.44457],[-1,3,-3,0],[9E+09,9E+09,9E+09,9E+09,9E+09,9E+09]];
    CONST robtarget rB_v13_t208_c2 := [[173.996,-336.828,2929.77],[0.770747,0.436735,0.13255,-0.44457],[0,0,-4,0],[9E+09,9E+09,9E+09,9E+09,9E+09,9E+09]];
    CONST robtarget rB_v13_t208_c5 := [[173.996,-336.828,2929.77],[0.770747,0.436735,0.13255,-0.44457],[0,0,0,0],[9E+09,9E+09,9E+09,9E+09,9E+09,9E+09]];
    CONST jointtarget jA_v13_t208 := [[-135.001,-18.0822,-7.61865,89.9994,55.3581,-180.001],[9E+09,9E+09,9E+09,9E+09,9E+09,9E+09]];
    CONST jointtarget jB_v13_t208 := [[-44.9991,-44.6077,-9.04692,270.001,43.5896,-269.999],[9E+09,9E+09,9E+09,9E+09,9E+09,9E+09]];
    CONST jointtarget jBseed_v13_t208 := [[-44.9991,-44.6077,-9.04691,270.001,43.5896,-269.999],[9E+09,9E+09,9E+09,9E+09,9E+09,9E+09]];

    CONST robtarget rA_v13_t210 := [[-0.0199233,-1505.01,1426],[0.117053,0.697354,-0.69735,0.117042],[-2,-1,1,0],[9E+09,9E+09,9E+09,9E+09,9E+09,9E+09]];
    CONST robtarget rB_v13_t210 := [[1899.63,-1805.19,274.9],[0.254994,0.805394,0.079064,0.529214],[-1,-3,-1,0],[9E+09,9E+09,9E+09,9E+09,9E+09,9E+09]];
    CONST robtarget rB_v13_t210_c5 := [[1899.63,-1805.19,274.9],[0.254994,0.805394,0.079064,0.529214],[0,0,0,0],[9E+09,9E+09,9E+09,9E+09,9E+09,9E+09]];
    CONST robtarget rB_v13_t210_c8 := [[1899.63,-1805.19,274.9],[0.254994,0.805394,0.079064,0.529214],[0,0,4,0],[9E+09,9E+09,9E+09,9E+09,9E+09,9E+09]];
    CONST jointtarget jA_v13_t210 := [[-90.0007,-22.3048,34.1661,-0.00069503,59.0826,179.999],[9E+09,9E+09,9E+09,9E+09,9E+09,9E+09]];
    CONST jointtarget jB_v13_t210 := [[-45.0004,56.195,-10.5585,-225,34.4523,-0.00042782],[9E+09,9E+09,9E+09,9E+09,9E+09,9E+09]];
    CONST jointtarget jBseed_v13_t210 := [[-45.0004,56.195,-10.5585,-225,34.4523,-0.000424055],[9E+09,9E+09,9E+09,9E+09,9E+09,9E+09]];

    CONST robtarget rA_v13_t211 := [[1899.63,-1805.19,274.9],[0.254994,0.805394,0.079064,0.529214],[-1,-3,-1,0],[9E+09,9E+09,9E+09,9E+09,9E+09,9E+09]];
    CONST robtarget rB_v13_t211 := [[-20.1035,-2928.29,1688.01],[0.472925,0.529167,0.464845,-0.52938],[-1,-1,-4,0],[9E+09,9E+09,9E+09,9E+09,9E+09,9E+09]];
    CONST robtarget rB_v13_t211_c5 := [[-20.1035,-2928.29,1688.01],[0.472925,0.529167,0.464845,-0.52938],[0,0,0,0],[9E+09,9E+09,9E+09,9E+09,9E+09,9E+09]];
    CONST jointtarget jA_v13_t211 := [[-45.0004,56.195,-10.5585,-225,34.4523,-0.00042782],[9E+09,9E+09,9E+09,9E+09,9E+09,9E+09]];
    CONST jointtarget jB_v13_t211 := [[-89.9993,56.4916,-63.9201,-44.9993,9.82024,-314.999],[9E+09,9E+09,9E+09,9E+09,9E+09,9E+09]];
    CONST jointtarget jBseed_v13_t211 := [[-89.9993,56.4916,-63.9201,-44.9993,9.82025,-314.999],[9E+09,9E+09,9E+09,9E+09,9E+09,9E+09]];

    CONST robtarget rA_v13_t212 := [[-20.1035,-2928.29,1688.01],[0.472925,0.529167,0.464845,-0.52938],[-1,-1,-4,0],[9E+09,9E+09,9E+09,9E+09,9E+09,9E+09]];
    CONST robtarget rB_v13_t212 := [[1796.88,-0.0173319,1860.47],[0.183287,-0.81101,0.335929,-0.442515],[-1,-1,-2,0],[9E+09,9E+09,9E+09,9E+09,9E+09,9E+09]];
    CONST robtarget rB_v13_t212_c2 := [[1796.88,-0.0173319,1860.47],[0.183287,-0.81101,0.335929,-0.442515],[0,0,-4,0],[9E+09,9E+09,9E+09,9E+09,9E+09,9E+09]];
    CONST jointtarget jA_v13_t212 := [[-89.9993,56.4916,-63.9201,-44.9993,9.82024,-314.999],[9E+09,9E+09,9E+09,9E+09,9E+09,9E+09]];
    CONST jointtarget jB_v13_t212 := [[-0.000526662,-10.9812,11.6709,-0.000526567,32.0737,-135.001],[9E+09,9E+09,9E+09,9E+09,9E+09,9E+09]];
    CONST jointtarget jBseed_v13_t212 := [[-0.000526658,-10.9812,11.6709,-0.000526658,32.0737,-135.001],[9E+09,9E+09,9E+09,9E+09,9E+09,9E+09]];

    CONST robtarget rA_v13_t213 := [[1796.88,-0.0173319,1860.47],[0.183287,-0.81101,0.335929,-0.442515],[-1,-1,-2,0],[9E+09,9E+09,9E+09,9E+09,9E+09,9E+09]];
    CONST robtarget rB_v13_t213 := [[1020.05,-1105.93,1796],[0.137952,-0.152205,0.702831,-0.681052],[-1,-2,3,0],[9E+09,9E+09,9E+09,9E+09,9E+09,9E+09]];
    CONST robtarget rB_v13_t213_c2 := [[1020.05,-1105.93,1796],[0.137952,-0.152205,0.702831,-0.681052],[0,0,-4,0],[9E+09,9E+09,9E+09,9E+09,9E+09,9E+09]];
    CONST robtarget rB_v13_t213_c5 := [[1020.05,-1105.93,1796],[0.137952,-0.152205,0.702831,-0.681052],[0,0,0,0],[9E+09,9E+09,9E+09,9E+09,9E+09,9E+09]];
    CONST jointtarget jA_v13_t213 := [[-0.000526662,-10.9812,11.6709,-0.000526567,32.0737,-135.001],[9E+09,9E+09,9E+09,9E+09,9E+09,9E+09]];
    CONST jointtarget jB_v13_t213 := [[-45.0009,-28.0105,30.1193,-90.0009,21.316,359.999],[9E+09,9E+09,9E+09,9E+09,9E+09,9E+09]];
    CONST jointtarget jBseed_v13_t213 := [[-45.0009,-28.0105,30.1193,-90.0009,21.316,359.999],[9E+09,9E+09,9E+09,9E+09,9E+09,9E+09]];

    CONST robtarget rA_v13_t217 := [[0.0068789,1700.52,1675.75],[0.438449,-0.55476,-0.554762,-0.438455],[0,-1,-3,0],[9E+09,9E+09,9E+09,9E+09,9E+09,9E+09]];
    CONST robtarget rB_v13_t217 := [[0.00335991,1053.06,2074.11],[0.830021,-0.405728,-0.16806,-0.343811],[0,1,-4,0],[9E+09,9E+09,9E+09,9E+09,9E+09,9E+09]];
    CONST robtarget rB_v13_t217_c1 := [[0.00335991,1053.06,2074.11],[0.830021,-0.405728,-0.16806,-0.343811],[0,-4,-4,0],[9E+09,9E+09,9E+09,9E+09,9E+09,9E+09]];
    CONST robtarget rB_v13_t217_c2 := [[0.00335991,1053.06,2074.11],[0.830021,-0.405728,-0.16806,-0.343811],[0,0,-4,0],[9E+09,9E+09,9E+09,9E+09,9E+09,9E+09]];
    CONST jointtarget jA_v13_t217 := [[89.9998,-17.7892,25.9655,-0.000250745,5.18204,-180],[9E+09,9E+09,9E+09,9E+09,9E+09,9E+09]];
    CONST jointtarget jB_v13_t217 := [[89.9998,-49.3905,35.2294,180,23.7385,-315],[9E+09,9E+09,9E+09,9E+09,9E+09,9E+09]];
    CONST jointtarget jBseed_v13_t217 := [[89.9998,-49.3905,35.2293,180,23.7385,-315],[9E+09,9E+09,9E+09,9E+09,9E+09,9E+09]];

    CONST robtarget rA_v13_t223 := [[2744.7,-11.5811,1170.86],[0.416215,0.599454,0.570589,0.376626],[-1,-1,-3,0],[9E+09,9E+09,9E+09,9E+09,9E+09,9E+09]];
    CONST robtarget rB_v13_t223 := [[-25.0252,-1961.79,2985.02],[0.630978,0.319185,0.220954,-0.67169],[-1,-1,1,0],[9E+09,9E+09,9E+09,9E+09,9E+09,9E+09]];
    CONST robtarget rB_v13_t223_c2 := [[-25.0252,-1961.79,2985.02],[0.630978,0.319185,0.220954,-0.67169],[0,0,-4,0],[9E+09,9E+09,9E+09,9E+09,9E+09,9E+09]];
    CONST robtarget rB_v13_t223_c3 := [[-25.0252,-1961.79,2985.02],[0.630978,0.319185,0.220954,-0.67169],[0,4,-4,0],[9E+09,9E+09,9E+09,9E+09,9E+09,9E+09]];
    CONST jointtarget jA_v13_t223 := [[-0.000519222,41.037,-23.2542,-45.0005,5.61602,-225.001],[9E+09,9E+09,9E+09,9E+09,9E+09,9E+09]];
    CONST jointtarget jB_v13_t223 := [[-89.9995,30.6656,-75.624,-89.9993,8.62453,90.0004],[9E+09,9E+09,9E+09,9E+09,9E+09,9E+09]];
    CONST jointtarget jBseed_v13_t223 := [[-89.9995,30.6656,-75.6239,-89.9995,8.62453,90.0005],[9E+09,9E+09,9E+09,9E+09,9E+09,9E+09]];

    CONST robtarget rA_v13_t226 := [[0.0287068,-1756.89,2046.15],[0.426928,0.563666,-0.563672,0.426951],[-1,0,-2,0],[9E+09,9E+09,9E+09,9E+09,9E+09,9E+09]];
    CONST robtarget rB_v13_t226 := [[-68.1767,-1026.5,3282.65],[0.6134,0.351773,0.0706954,-0.703561],[-1,-1,-3,0],[9E+09,9E+09,9E+09,9E+09,9E+09,9E+09]];
    CONST robtarget rB_v13_t226_c2 := [[-68.1767,-1026.5,3282.65],[0.6134,0.351773,0.0706954,-0.703561],[0,0,-4,0],[9E+09,9E+09,9E+09,9E+09,9E+09,9E+09]];
    CONST robtarget rB_v13_t226_c3 := [[-68.1767,-1026.5,3282.65],[0.6134,0.351773,0.0706954,-0.703561],[0,4,-4,0],[9E+09,9E+09,9E+09,9E+09,9E+09,9E+09]];
    CONST jointtarget jA_v13_t226 := [[-89.9991,-12.8489,8.02484,0.000905057,20.5414,-179.999],[9E+09,9E+09,9E+09,9E+09,9E+09,9E+09]];
    CONST jointtarget jB_v13_t226 := [[-89.9998,-6.13605,-48.2925,-89.9999,24.0956,-270],[9E+09,9E+09,9E+09,9E+09,9E+09,9E+09]];
    CONST jointtarget jBseed_v13_t226 := [[-89.9998,-6.13605,-48.2925,-89.9998,24.0956,-270],[9E+09,9E+09,9E+09,9E+09,9E+09,9E+09]];

